KUKA KRL program: EPS_2_25694_LG01A_A_20260223033035.src

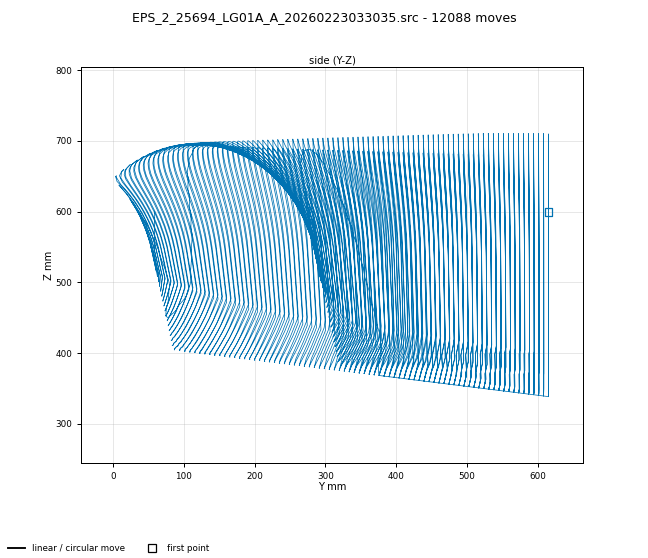
[picture p0: tool path of EPS_2_25694_LG01A_A_20260223033035.src, 12088 of 12090 moves have a stored position in this frame; points joined in program order, loops and branches not executed]
&ACCESS RVP
&REL 4
&COMMENT QRS 19112012
&PARAM EDITMASK = *
DEF PART()
EXT BAS (BAS_COMMAND :IN,REAL :IN )
INT I
BAS (#INITMOV,0 )

;KUKA QRS Post kuka4.cps  Date:22-06-2017 !

File_ID=3040

QRS_PRE_INIT()

;Init var - Until changes are made in qrs_pre_init
Outlet_Square_prg=0
Inlet_1_Square_prg=0
Inlet_2_Square_prg=0
Inlet_3_Square_prg=0
Inlet_4_Square_prg=0
Inlet_5_Square_prg=0

Outlet_1={X 0.000, Y 517.920, Z 561.000, B 0.000, E1 0.000 }
Inlet_1={X 0.000, Y 520.110, Z 531.000, B 0.000, E1 251.000 }
Outlet_1_type=299
Inlet_1_type=299
;QRS#1=Sidecore dimensions
;QRS#2=300-12" PVC SDR 35
;QRS#3=300-12" PVC SDR 35
;QRS#4=
;QRS#5=
;QRS#6=
;QRS#7=
;QRS#8=
;QRS#9=16M PSX
;QRS#10=16M PSX
;QRS#11=
;QRS#12=
;QRS#13=
;QRS#14=
;QRS#15=
;QRS#16=1220x127x991 3,25'
;QRS#17=EPS Height
;QRS#18=710,5
;QRS#19=*
;QRS#20= UPDATED VERSION 22-06-2017
;QRS#21=*
Outlet_Square=0150
Inlet_1_Square=0150
Inlet_2_Square=0
Inlet_3_Square=0
Inlet_4_Square=0
Inlet_5_Square=0
Mill_Square=1
Outlet_Square_Prg=206
Inlet_1_Square_prg=206

QRS_INIT()

$ADVANCE=5

; T1
PTP {E1 173.642,E2 173.642}
PTP {X 0,Y 615.447,A -85,B 0,C 180,E1 173.642,E2 173.642,E3 0,E4 0,E5 0,E6 0}
QRS_SPEED_INIT()
LIN {X 0,Y 615.447,Z 600,A -85,B 0,C 180,E1 173.642,E2 173.642,E3 0,E4 0,E5 0,E6 0} C_VEL
LIN {X 0,Y 615.447,Z 348.502,A -85,B 0,C 180,E1 173.642,E2 173.642} C_VEL
LIN {X 0,Y 615.447,Z 340.324,A -85,B 0,C 180,E1 173.642,E2 173.642} C_VEL
LIN {X 0,Y 615.428,Z 338.324,A -85,B 0,C 180,E1 173.456,E2 173.456} C_VEL
LIN {X 0,Y 615.429,Z 338.324,A -85,B 0,C 180,E1 171.462,E2 171.462} C_VEL
LIN {X 0,Y 615.412,Z 338.324,A -85,B 0,C 180,E1 169.14,E2 169.14} C_VEL
LIN {X 0,Y 615.415,Z 338.325,A -85,B 0,C 180,E1 166.797,E2 166.797} C_VEL
LIN {X 0,Y 615.418,Z 338.324,A -85,B 0,C 180,E1 164.772,E2 164.772} C_VEL
LIN {X 0,Y 615.493,Z 338.326,A -85,B 0,C 180,E1 162.043,E2 162.043} C_VEL
LIN {X 0,Y 615.419,Z 338.323,A -85,B 0,C 180,E1 159.267,E2 159.267} C_VEL
LIN {X 0,Y 615.416,Z 338.323,A -85,B 0,C 180,E1 157.152,E2 157.152} C_VEL
LIN {X 0,Y 615.416,Z 338.323,A -85,B 0,C 180,E1 155.005,E2 155.005} C_VEL
LIN {X 0,Y 615.478,Z 338.329,A -85,B 0,C 180,E1 152.084,E2 152.084} C_VEL
LIN {X 0,Y 615.475,Z 338.321,A -85,B 0,C 180,E1 149.839,E2 149.839} C_VEL
LIN {X 0,Y 615.44,Z 338.322,A -85,B 0,C 180,E1 147.539,E2 147.539} C_VEL
LIN {X 0,Y 615.42,Z 338.322,A -85,B 0,C 180,E1 145.18,E2 145.18} C_VEL
LIN {X 0,Y 615.429,Z 338.323,A -85,B 0,C 180,E1 142.753,E2 142.753} C_VEL
LIN {X 0,Y 615.486,Z 338.32,A -85,B 0,C 180,E1 139.909,E2 139.909} C_VEL
LIN {X 0,Y 615.451,Z 338.32,A -85,B 0,C 180,E1 137.644,E2 137.644} C_VEL
LIN {X 0,Y 615.422,Z 338.322,A -85,B 0,C 180,E1 135.073,E2 135.073} C_VEL
LIN {X 0,Y 615.423,Z 338.322,A -85,B 0,C 180,E1 133.041,E2 133.041} C_VEL
LIN {X 0,Y 615.446,Z 338.323,A -85,B 0,C 180,E1 130.608,E2 130.608} C_VEL
LIN {X 0,Y 615.484,Z 338.322,A -85,B 0,C 180,E1 128.011,E2 128.011} C_VEL
LIN {X 0,Y 615.45,Z 338.319,A -85,B 0,C 180,E1 125.617,E2 125.617} C_VEL
LIN {X 0,Y 615.428,Z 338.32,A -85,B 0,C 180,E1 123.238,E2 123.238} C_VEL
LIN {X 0,Y 615.43,Z 338.322,A -85,B 0,C 180,E1 120.921,E2 120.921} C_VEL
LIN {X 0,Y 615.468,Z 338.325,A -85,B 0,C 180,E1 118.446,E2 118.446} C_VEL
LIN {X 0,Y 615.447,Z 338.318,A -85,B 0,C 180,E1 115.56,E2 115.56} C_VEL
LIN {X 0,Y 615.447,Z 338.318,A -85,B 0,C 180,E1 113.557,E2 113.557} C_VEL
LIN {X 0,Y 615.439,Z 338.319,A -85,B 0,C 180,E1 111.432,E2 111.432} C_VEL
LIN {X 0,Y 615.435,Z 338.319,A -85,B 0,C 180,E1 109.338,E2 109.338} C_VEL
LIN {X 0,Y 615.431,Z 338.32,A -85,B 0,C 180,E1 107.271,E2 107.271} C_VEL
LIN {X 0,Y 615.433,Z 338.319,A -85,B 0,C 180,E1 105.226,E2 105.226} C_VEL
LIN {X 0,Y 615.433,Z 338.32,A -85,B 0,C 180,E1 103.201,E2 103.201} C_VEL
LIN {X 0,Y 615.47,Z 338.324,A -85,B 0,C 180,E1 100.526,E2 100.526} C_VEL
LIN {X 0,Y 615.48,Z 338.315,A -85,B 0,C 180,E1 97.875,E2 97.875} C_VEL
LIN {X 0,Y 615.436,Z 338.319,A -85,B 0,C 180,E1 95.241,E2 95.241} C_VEL
LIN {X 0,Y 615.464,Z 338.323,A -85,B 0,C 180,E1 92.617,E2 92.617} C_VEL
LIN {X 0,Y 615.486,Z 338.316,A -85,B 0,C 180,E1 89.999,E2 89.999} C_VEL
LIN {X 0,Y 615.441,Z 338.317,A -85,B 0,C 180,E1 87.381,E2 87.381} C_VEL
LIN {X 0,Y 615.443,Z 338.317,A -85,B 0,C 180,E1 85.414,E2 85.414} C_VEL
LIN {X 0,Y 615.445,Z 338.317,A -85,B 0,C 180,E1 83.442,E2 83.442} C_VEL
LIN {X 0,Y 615.446,Z 338.316,A -85,B 0,C 180,E1 81.462,E2 81.462} C_VEL
LIN {X 0,Y 615.44,Z 338.319,A -85,B 0,C 180,E1 79.137,E2 79.137} C_VEL
LIN {X 0,Y 615.455,Z 338.322,A -85,B 0,C 180,E1 76.797,E2 76.797} C_VEL
LIN {X 0,Y 615.494,Z 338.315,A -85,B 0,C 180,E1 74.094,E2 74.094} C_VEL
LIN {X 0,Y 615.444,Z 338.317,A -85,B 0,C 180,E1 71.352,E2 71.352} C_VEL
LIN {X 0,Y 615.443,Z 338.318,A -85,B 0,C 180,E1 69.267,E2 69.267} C_VEL
LIN {X 0,Y 615.444,Z 338.319,A -85,B 0,C 180,E1 67.153,E2 67.153} C_VEL
LIN {X 0,Y 615.499,Z 338.325,A -85,B 0,C 180,E1 64.43,E2 64.43} C_VEL
LIN {X 0,Y 615.455,Z 338.315,A -85,B 0,C 180,E1 61.556,E2 61.556} C_VEL
LIN {X 0,Y 615.445,Z 338.32,A -85,B 0,C 180,E1 59.077,E2 59.077} C_VEL
LIN {X 0,Y 615.497,Z 338.325,A -85,B 0,C 180,E1 56.465,E2 56.465} C_VEL
LIN {X 0,Y 615.457,Z 338.314,A -85,B 0,C 180,E1 53.572,E2 53.572} C_VEL
LIN {X 0,Y 615.456,Z 338.32,A -85,B 0,C 180,E1 50.942,E2 50.942} C_VEL
LIN {X 0,Y 615.493,Z 338.326,A -85,B 0,C 180,E1 48.526,E2 48.526} C_VEL
LIN {X 0,Y 615.482,Z 338.311,A -85,B 0,C 180,E1 45.849,E2 45.849} C_VEL
LIN {X 0,Y 615.45,Z 338.317,A -85,B 0,C 180,E1 43.248,E2 43.248} C_VEL
LIN {X 0,Y 615.449,Z 338.397,A -85,B 0,C 180,E1 41.259,E2 41.259} C_VEL
LIN {X 0,Y 615.47,Z 358.127,A -85,B 0,C 180,E1 38.696,E2 38.696} C_VEL
LIN {X 0,Y 615.456,Z 369.9,A -85,B 0,C 180,E1 37.186,E2 37.186} C_VEL
LIN {X 0,Y 615.489,Z 534.997,A -85,B 0,C 180,E1 35.19,E2 35.19} C_VEL
LIN {X 0,Y 615.484,Z 550.512,A -85,B 0,C 180,E1 34.865,E2 34.865} C_VEL
LIN {X 0,Y 615.478,Z 565.792,A -85,B 0,C 180,E1 34.402,E2 34.402} C_VEL
LIN {X 0,Y 615.484,Z 579.854,A -85,B 0,C 180,E1 33.838,E2 33.838} C_VEL
LIN {X 0,Y 615.488,Z 593.728,A -85,B 0,C 180,E1 33.139,E2 33.139} C_VEL
LIN {X 0,Y 615.498,Z 606.785,A -85,B 0,C 180,E1 32.332,E2 32.332} C_VEL
LIN {X 0,Y 615.496,Z 619.457,A -85,B 0,C 180,E1 31.385,E2 31.385} C_VEL
LIN {X 0,Y 615.494,Z 631.006,A -85,B 0,C 180,E1 30.349,E2 30.349} C_VEL
LIN {X 0,Y 615.494,Z 641.505,A -85,B 0,C 180,E1 29.219,E2 29.219} C_VEL
LIN {X 0,Y 615.496,Z 649.597,A -85,B 0,C 180,E1 28.182,E2 28.182} C_VEL
LIN {X 0,Y 615.493,Z 657.085,A -85,B 0,C 180,E1 27.045,E2 27.045} C_VEL
LIN {X 0,Y 615.499,Z 664.276,A -85,B 0,C 180,E1 25.715,E2 25.715} C_VEL
LIN {X 0,Y 615.488,Z 669.041,A -85,B 0,C 180,E1 24.632,E2 24.632} C_VEL
LIN {X 0,Y 615.491,Z 672.806,A -85,B 0,C 180,E1 23.556,E2 23.556} C_VEL
LIN {X 0,Y 615.496,Z 676.516,A -85,B 0,C 180,E1 22.136,E2 22.136} C_VEL
LIN {X 0,Y 615.495,Z 678.815,A -85,B 0,C 180,E1 20.731,E2 20.731} C_VEL
LIN {X 0,Y 615.489,Z 679.804,A -85,B 0,C 180,E1 19.338,E2 19.338} C_VEL
LIN {X 0,Y 615.497,Z 679.524,A -85,B 0,C 180,E1 17.957,E2 17.957} C_VEL
LIN {X 0,Y 615.493,Z 677.757,A -85,B 0,C 180,E1 16.432,E2 16.432} C_VEL
LIN {X 0,Y 615.492,Z 675.277,A -85,B 0,C 180,E1 15.226,E2 15.226} C_VEL
LIN {X 0,Y 615.495,Z 671.262,A -85,B 0,C 180,E1 13.874,E2 13.874} C_VEL
LIN {X 0,Y 615.492,Z 665.885,A -85,B 0,C 180,E1 12.53,E2 12.53} C_VEL
LIN {X 0,Y 615.496,Z 659.043,A -85,B 0,C 180,E1 11.193,E2 11.193} C_VEL
LIN {X 0,Y 615.496,Z 650.583,A -85,B 0,C 180,E1 9.862,E2 9.862} C_VEL
LIN {X 0,Y 615.495,Z 641.592,A -85,B 0,C 180,E1 8.702,E2 8.702} C_VEL
LIN {X 0,Y 615.494,Z 630.85,A -85,B 0,C 180,E1 7.546,E2 7.546} C_VEL
LIN {X 0,Y 615.498,Z 619.859,A -85,B 0,C 180,E1 6.557,E2 6.557} C_VEL
LIN {X 0,Y 615.498,Z 607.894,A -85,B 0,C 180,E1 5.652,E2 5.652} C_VEL
LIN {X 0,Y 615.492,Z 594.819,A -85,B 0,C 180,E1 4.831,E2 4.831} C_VEL
LIN {X 0,Y 615.493,Z 580.329,A -85,B 0,C 180,E1 4.093,E2 4.093} C_VEL
LIN {X 0,Y 615.478,Z 566.113,A -85,B 0,C 180,E1 3.519,E2 3.519} C_VEL
LIN {X 0,Y 615.484,Z 551.397,A -85,B 0,C 180,E1 3.068,E2 3.068} C_VEL
LIN {X 0,Y 615.49,Z 536.141,A -85,B 0,C 180,E1 2.741,E2 2.741} C_VEL
LIN {X 0,Y 615.483,Z 493.536,A -85,B 0,C 180,E1 2.209,E2 2.209} C_VEL
LIN {X 0,Y 615.457,Z 369.836,A -85,B 0,C 180,E1 0.716,E2 0.716} C_VEL
LIN {X 0,Y 615.49,Z 347.76,A -85,B 0,C 180,E1 -2.127,E2 -2.127} C_VEL
LIN {X 0,Y 615.457,Z 338.316,A -85,B 0,C 180,E1 -3.375,E2 -3.375} C_VEL
LIN {X 0,Y 615.487,Z 338.31,A -85,B 0,C 180,E1 -5.898,E2 -5.898} C_VEL
LIN {X 0,Y 615.489,Z 338.327,A -85,B 0,C 180,E1 -8.536,E2 -8.536} C_VEL
LIN {X 0,Y 615.449,Z 338.318,A -85,B 0,C 180,E1 -11.194,E2 -11.194} C_VEL
LIN {X 0,Y 615.491,Z 338.311,A -85,B 0,C 180,E1 -13.933,E2 -13.933} C_VEL
LIN {X 0,Y 615.476,Z 338.325,A -85,B 0,C 180,E1 -16.587,E2 -16.587} C_VEL
LIN {X 0,Y 615.47,Z 338.323,A -85,B 0,C 180,E1 -18.646,E2 -18.646} C_VEL
LIN {X 0,Y 615.458,Z 338.322,A -85,B 0,C 180,E1 -20.732,E2 -20.732} C_VEL
LIN {X 0,Y 615.447,Z 338.322,A -85,B 0,C 180,E1 -22.846,E2 -22.846} C_VEL
LIN {X 0,Y 615.437,Z 338.321,A -85,B 0,C 180,E1 -24.994,E2 -24.994} C_VEL
LIN {X 0,Y 615.432,Z 338.32,A -85,B 0,C 180,E1 -27.18,E2 -27.18} C_VEL
LIN {X 0,Y 615.471,Z 338.317,A -85,B 0,C 180,E1 -29.791,E2 -29.791} C_VEL
LIN {X 0,Y 615.465,Z 338.324,A -85,B 0,C 180,E1 -32.459,E2 -32.459} C_VEL
LIN {X 0,Y 615.43,Z 338.323,A -85,B 0,C 180,E1 -34.819,E2 -34.819} C_VEL
LIN {X 0,Y 615.423,Z 338.322,A -85,B 0,C 180,E1 -37.247,E2 -37.247} C_VEL
LIN {X 0,Y 615.498,Z 338.325,A -85,B 0,C 180,E1 -40.089,E2 -40.089} C_VEL
LIN {X 0,Y 615.457,Z 338.325,A -85,B 0,C 180,E1 -42.355,E2 -42.355} C_VEL
LIN {X 0,Y 615.412,Z 338.325,A -85,B 0,C 180,E1 -44.924,E2 -44.924} C_VEL
LIN {X 0,Y 615.41,Z 338.325,A -85,B 0,C 180,E1 -46.96,E2 -46.96} C_VEL
LIN {X 0,Y 615.426,Z 338.325,A -85,B 0,C 180,E1 -49.388,E2 -49.388} C_VEL
LIN {X 0,Y 615.477,Z 338.328,A -85,B 0,C 180,E1 -51.989,E2 -51.989} C_VEL
LIN {X 0,Y 615.447,Z 338.322,A -85,B 0,C 180,E1 -54.381,E2 -54.381} C_VEL
LIN {X 0,Y 615.423,Z 338.322,A -85,B 0,C 180,E1 -56.759,E2 -56.759} C_VEL
LIN {X 0,Y 615.423,Z 338.323,A -85,B 0,C 180,E1 -59.076,E2 -59.076} C_VEL
LIN {X 0,Y 615.466,Z 338.324,A -85,B 0,C 180,E1 -61.553,E2 -61.553} C_VEL
LIN {X 0,Y 615.447,Z 338.319,A -85,B 0,C 180,E1 -64.439,E2 -64.439} C_VEL
LIN {X 0,Y 615.43,Z 338.439,A -85,B 0,C 180,E1 -64.934,E2 -64.934} C_VEL
LIN {X 0,Y 615.477,Z 359.979,A -85,B 0,C 180,E1 -67.404,E2 -67.404} C_VEL
LIN {X 0,Y 615.49,Z 384.309,A -85,B 0,C 180,E1 -70.141,E2 -70.141} C_VEL
LIN {X 0,Y 615.487,Z 398.969,A -85,B 0,C 180,E1 -71.761,E2 -71.761} C_VEL
LIN {X 0,Y 615.484,Z 565.198,A -85,B 0,C 180,E1 -73.768,E2 -73.768} C_VEL
LIN {X 0,Y 615.49,Z 580.682,A -85,B 0,C 180,E1 -74.094,E2 -74.094} C_VEL
LIN {X 0,Y 615.48,Z 596.028,A -85,B 0,C 180,E1 -74.561,E2 -74.561} C_VEL
LIN {X 0,Y 615.484,Z 609.735,A -85,B 0,C 180,E1 -75.112,E2 -75.112} C_VEL
LIN {X 0,Y 615.493,Z 624.04,A -85,B 0,C 180,E1 -75.833,E2 -75.833} C_VEL
LIN {X 0,Y 615.497,Z 636.886,A -85,B 0,C 180,E1 -76.63,E2 -76.63} C_VEL
LIN {X 0,Y 615.495,Z 649.244,A -85,B 0,C 180,E1 -77.553,E2 -77.553} C_VEL
LIN {X 0,Y 615.495,Z 659.598,A -85,B 0,C 180,E1 -78.473,E2 -78.473} C_VEL
LIN {X 0,Y 615.494,Z 669.176,A -85,B 0,C 180,E1 -79.472,E2 -79.472} C_VEL
LIN {X 0,Y 615.493,Z 678.571,A -85,B 0,C 180,E1 -80.635,E2 -80.635} C_VEL
LIN {X 0,Y 615.497,Z 686.375,A -85,B 0,C 180,E1 -81.793,E2 -81.793} C_VEL
LIN {X 0,Y 615.494,Z 693.607,A -85,B 0,C 180,E1 -83.102,E2 -83.102} C_VEL
LIN {X 0,Y 615.499,Z 699.433,A -85,B 0,C 180,E1 -84.429,E2 -84.429} C_VEL
LIN {X 0,Y 615.491,Z 702.857,A -85,B 0,C 180,E1 -85.415,E2 -85.415} C_VEL
LIN {X 0,Y 615.493,Z 706.316,A -85,B 0,C 180,E1 -86.726,E2 -86.726} C_VEL
LIN {X 0,Y 615.499,Z 708.592,A -85,B 0,C 180,E1 -88.036,E2 -88.036} C_VEL
LIN {X 0,Y 615.491,Z 709.741,A -85,B 0,C 180,E1 -89.345,E2 -89.345} C_VEL
LIN {X 0,Y 615.491,Z 709.741,A -85,B 0,C 180,E1 -90.653,E2 -90.653} C_VEL
LIN {X 0,Y 615.499,Z 708.594,A -85,B 0,C 180,E1 -91.962,E2 -91.962} C_VEL
LIN {X 0,Y 615.493,Z 706.32,A -85,B 0,C 180,E1 -93.272,E2 -93.272} C_VEL
LIN {X 0,Y 615.491,Z 702.863,A -85,B 0,C 180,E1 -94.583,E2 -94.583} C_VEL
LIN {X 0,Y 615.497,Z 698.147,A -85,B 0,C 180,E1 -95.897,E2 -95.897} C_VEL
LIN {X 0,Y 615.492,Z 692.035,A -85,B 0,C 180,E1 -97.215,E2 -97.215} C_VEL
LIN {X 0,Y 615.49,Z 684.34,A -85,B 0,C 180,E1 -98.536,E2 -98.536} C_VEL
LIN {X 0,Y 615.495,Z 676.122,A -85,B 0,C 180,E1 -99.695,E2 -99.695} C_VEL
LIN {X 0,Y 615.496,Z 665.899,A -85,B 0,C 180,E1 -100.892,E2 -100.892} C_VEL
LIN {X 0,Y 615.496,Z 656.079,A -85,B 0,C 180,E1 -101.859,E2 -101.859} C_VEL
LIN {X 0,Y 615.497,Z 643.963,A -85,B 0,C 180,E1 -102.864,E2 -102.864} C_VEL
LIN {X 0,Y 615.498,Z 631.815,A -85,B 0,C 180,E1 -103.704,E2 -103.704} C_VEL
LIN {X 0,Y 615.477,Z 618.398,A -85,B 0,C 180,E1 -104.472,E2 -104.472} C_VEL
LIN {X 0,Y 615.495,Z 603.875,A -85,B 0,C 180,E1 -105.14,E2 -105.14} C_VEL
LIN {X 0,Y 615.48,Z 589.652,A -85,B 0,C 180,E1 -105.649,E2 -105.649} C_VEL
LIN {X 0,Y 615.5,Z 575.193,A -85,B 0,C 180,E1 -106.034,E2 -106.034} C_VEL
LIN {X 0,Y 615.48,Z 560.694,A -85,B 0,C 180,E1 -106.296,E2 -106.296} C_VEL
LIN {X 0,Y 615.489,Z 398.746,A -85,B 0,C 180,E1 -108.258,E2 -108.258} C_VEL
LIN {X 0,Y 615.49,Z 373.403,A -85,B 0,C 180,E1 -111.079,E2 -111.079} C_VEL
LIN {X 0,Y 615.496,Z 347.578,A -85,B 0,C 180,E1 -114.01,E2 -114.01} C_VEL
LIN {X 0,Y 615.43,Z 338.321,A -85,B 0,C 180,E1 -115.099,E2 -115.099} C_VEL
LIN {X 0,Y 615.429,Z 338.32,A -85,B 0,C 180,E1 -117.179,E2 -117.179} C_VEL
LIN {X 0,Y 615.47,Z 338.317,A -85,B 0,C 180,E1 -119.792,E2 -119.792} C_VEL
LIN {X 0,Y 615.468,Z 338.324,A -85,B 0,C 180,E1 -122.457,E2 -122.457} C_VEL
LIN {X 0,Y 615.435,Z 338.322,A -85,B 0,C 180,E1 -124.817,E2 -124.817} C_VEL
LIN {X 0,Y 615.428,Z 338.32,A -85,B 0,C 180,E1 -127.245,E2 -127.245} C_VEL
LIN {X 0,Y 615.499,Z 338.321,A -85,B 0,C 180,E1 -130.09,E2 -130.09} C_VEL
LIN {X 0,Y 615.476,Z 338.324,A -85,B 0,C 180,E1 -132.352,E2 -132.352} C_VEL
LIN {X 0,Y 615.426,Z 338.322,A -85,B 0,C 180,E1 -134.926,E2 -134.926} C_VEL
LIN {X 0,Y 615.425,Z 338.322,A -85,B 0,C 180,E1 -136.957,E2 -136.957} C_VEL
LIN {X 0,Y 615.431,Z 338.321,A -85,B 0,C 180,E1 -139.389,E2 -139.389} C_VEL
LIN {X 0,Y 615.478,Z 338.324,A -85,B 0,C 180,E1 -141.987,E2 -141.987} C_VEL
LIN {X 0,Y 615.465,Z 338.324,A -85,B 0,C 180,E1 -144.383,E2 -144.383} C_VEL
LIN {X 0,Y 615.429,Z 338.323,A -85,B 0,C 180,E1 -146.76,E2 -146.76} C_VEL
LIN {X 0,Y 615.419,Z 338.323,A -85,B 0,C 180,E1 -149.077,E2 -149.077} C_VEL
LIN {X 0,Y 615.425,Z 338.322,A -85,B 0,C 180,E1 -151.339,E2 -151.339} C_VEL
LIN {X 0,Y 615.472,Z 338.325,A -85,B 0,C 180,E1 -154.284,E2 -154.284} C_VEL
LIN {X 0,Y 615.451,Z 338.324,A -85,B 0,C 180,E1 -156.442,E2 -156.442} C_VEL
LIN {X 0,Y 615.437,Z 338.324,A -85,B 0,C 180,E1 -158.566,E2 -158.566} C_VEL
LIN {X 0,Y 615.429,Z 338.324,A -85,B 0,C 180,E1 -160.66,E2 -160.66} C_VEL
LIN {X 0,Y 615.423,Z 338.324,A -85,B 0,C 180,E1 -162.728,E2 -162.728} C_VEL
LIN {X 0,Y 615.42,Z 338.324,A -85,B 0,C 180,E1 -164.772,E2 -164.772} C_VEL
LIN {X 0,Y 615.416,Z 338.325,A -85,B 0,C 180,E1 -166.797,E2 -166.797} C_VEL
LIN {X 0,Y 615.413,Z 338.324,A -85,B 0,C 180,E1 -169.139,E2 -169.139} C_VEL
LIN {X 0,Y 615.429,Z 338.324,A -85,B 0,C 180,E1 -171.463,E2 -171.463} C_VEL
LIN {X 0,Y 615.485,Z 338.326,A -85,B 0,C 180,E1 -174.102,E2 -174.102} C_VEL
LIN {X 0,Y 615.417,Z 338.325,A -85,B 0,C 180,E1 -176.727,E2 -176.727} C_VEL
LIN {X 0,Y 615.418,Z 338.325,A -85,B 0,C 180,E1 -178.691,E2 -178.691} C_VEL
LIN {X 0,Y 615.419,Z 338.325,A -85,B 0,C 180,E1 -180.655,E2 -180.655} C_VEL
LIN {X 0,Y 615.421,Z 338.325,A -85,B 0,C 180,E1 -182.618,E2 -182.618} C_VEL
LIN {X 0,Y 615.424,Z 338.325,A -85,B 0,C 180,E1 -184.585,E2 -184.585} C_VEL
LIN {X 0,Y 615.428,Z 338.324,A -85,B 0,C 180,E1 -186.544,E2 -186.544} C_VEL
LIN {X 0,Y 614.74,Z 338.47,A -85,B 0,C 180,E1 -187.09,E2 -187.09} C_VEL
LIN {X 0,Y 611.894,Z 338.895,A -85,B 0,C 180,E1 -187.976,E2 -187.976} C_VEL
LIN {X 0,Y 609.509,Z 339.197,A -85,B 0,C 180,E1 -188.689,E2 -188.689} C_VEL
LIN {X 0,Y 608.491,Z 339.31,A -85,B 0,C 180,E1 -189.239,E2 -189.239} C_VEL
LIN {X 0,Y 608.411,Z 339.319,A -85,B 0,C 180,E1 -189.425,E2 -189.425} C_VEL
LIN {X 0,Y 608.443,Z 339.324,A -85,B 0,C 180,E1 -192,E2 -192} C_VEL
LIN {X 0,Y 608.389,Z 339.321,A -85,B 0,C 180,E1 -194.723,E2 -194.723} C_VEL
LIN {X 0,Y 608.397,Z 339.319,A -85,B 0,C 180,E1 -196.786,E2 -196.786} C_VEL
LIN {X 0,Y 608.412,Z 339.317,A -85,B 0,C 180,E1 -198.871,E2 -198.871} C_VEL
LIN {X 0,Y 608.436,Z 339.321,A -85,B 0,C 180,E1 -201.693,E2 -201.693} C_VEL
LIN {X 0,Y 608.412,Z 339.318,A -85,B 0,C 180,E1 -204.573,E2 -204.573} C_VEL
LIN {X 0,Y 608.402,Z 339.319,A -85,B 0,C 180,E1 -207.197,E2 -207.197} C_VEL
LIN {X 0,Y 608.462,Z 339.32,A -85,B 0,C 180,E1 -209.974,E2 -209.974} C_VEL
LIN {X 0,Y 608.411,Z 339.317,A -85,B 0,C 180,E1 -212.883,E2 -212.883} C_VEL
LIN {X 0,Y 608.406,Z 339.32,A -85,B 0,C 180,E1 -215.28,E2 -215.28} C_VEL
LIN {X 0,Y 608.451,Z 339.317,A -85,B 0,C 180,E1 -218.241,E2 -218.241} C_VEL
LIN {X 0,Y 608.399,Z 339.32,A -85,B 0,C 180,E1 -221.182,E2 -221.182} C_VEL
LIN {X 0,Y 608.461,Z 339.322,A -85,B 0,C 180,E1 -223.871,E2 -223.871} C_VEL
LIN {X 0,Y 608.421,Z 339.316,A -85,B 0,C 180,E1 -226.697,E2 -226.697} C_VEL
LIN {X 0,Y 608.396,Z 339.319,A -85,B 0,C 180,E1 -228.82,E2 -228.82} C_VEL
LIN {X 0,Y 608.46,Z 339.322,A -85,B 0,C 180,E1 -231.761,E2 -231.761} C_VEL
LIN {X 0,Y 608.405,Z 339.318,A -85,B 0,C 180,E1 -234.722,E2 -234.722} C_VEL
LIN {X 0,Y 608.443,Z 339.319,A -85,B 0,C 180,E1 -237.481,E2 -237.481} C_VEL
LIN {X 0,Y 608.456,Z 339.315,A -85,B 0,C 180,E1 -240.221,E2 -240.221} C_VEL
LIN {X 0,Y 608.411,Z 339.317,A -85,B 0,C 180,E1 -242.806,E2 -242.806} C_VEL
LIN {X 0,Y 608.432,Z 339.32,A -85,B 0,C 180,E1 -245.429,E2 -245.429} C_VEL
LIN {X 0,Y 608.445,Z 339.315,A -85,B 0,C 180,E1 -248.309,E2 -248.309} C_VEL
LIN {X 0,Y 608.432,Z 339.316,A -85,B 0,C 180,E1 -251.131,E2 -251.131} C_VEL
LIN {X 0,Y 608.455,Z 339.319,A -85,B 0,C 180,E1 -253.907,E2 -253.907} C_VEL
LIN {X 0,Y 608.425,Z 339.316,A -85,B 0,C 180,E1 -256.644,E2 -256.644} C_VEL
LIN {X 0,Y 608.439,Z 339.319,A -85,B 0,C 180,E1 -259.351,E2 -259.351} C_VEL
LIN {X 0,Y 608.472,Z 339.315,A -85,B 0,C 180,E1 -262.034,E2 -262.034} C_VEL
LIN {X 0,Y 608.422,Z 339.316,A -85,B 0,C 180,E1 -264.699,E2 -264.699} C_VEL
LIN {X 0,Y 608.456,Z 339.317,A -85,B 0,C 180,E1 -267.353,E2 -267.353} C_VEL
LIN {X 0,Y 608.477,Z 339.314,A -85,B 0,C 180,E1 -270.001,E2 -270.001} C_VEL
LIN {X 0,Y 608.437,Z 339.314,A -85,B 0,C 180,E1 -272.649,E2 -272.649} C_VEL
LIN {X 0,Y 608.44,Z 339.319,A -85,B 0,C 180,E1 -275.303,E2 -275.303} C_VEL
LIN {X 0,Y 608.481,Z 339.313,A -85,B 0,C 180,E1 -277.968,E2 -277.968} C_VEL
LIN {X 0,Y 608.412,Z 339.318,A -85,B 0,C 180,E1 -280.926,E2 -280.926} C_VEL
LIN {X 0,Y 608.444,Z 339.32,A -85,B 0,C 180,E1 -283.358,E2 -283.358} C_VEL
LIN {X 0,Y 608.454,Z 339.315,A -85,B 0,C 180,E1 -286.095,E2 -286.095} C_VEL
LIN {X 0,Y 608.438,Z 339.315,A -85,B 0,C 180,E1 -288.871,E2 -288.871} C_VEL
LIN {X 0,Y 608.466,Z 339.319,A -85,B 0,C 180,E1 -291.692,E2 -291.692} C_VEL
LIN {X 0,Y 608.431,Z 339.315,A -85,B 0,C 180,E1 -294.573,E2 -294.573} C_VEL
LIN {X 0,Y 608.456,Z 339.316,A -85,B 0,C 180,E1 -297.202,E2 -297.202} C_VEL
LIN {X 0,Y 608.471,Z 339.313,A -85,B 0,C 180,E1 -299.971,E2 -299.971} C_VEL
LIN {X 0,Y 608.438,Z 339.315,A -85,B 0,C 180,E1 -302.881,E2 -302.881} C_VEL
LIN {X 0,Y 608.435,Z 339.321,A -85,B 0,C 180,E1 -305.279,E2 -305.279} C_VEL
LIN {X 0,Y 608.461,Z 339.312,A -85,B 0,C 180,E1 -308.239,E2 -308.239} C_VEL
LIN {X 0,Y 608.436,Z 339.32,A -85,B 0,C 180,E1 -311.179,E2 -311.179} C_VEL
LIN {X 0,Y 608.469,Z 339.314,A -85,B 0,C 180,E1 -313.87,E2 -313.87} C_VEL
LIN {X 0,Y 608.443,Z 339.314,A -85,B 0,C 180,E1 -316.695,E2 -316.695} C_VEL
LIN {X 0,Y 608.452,Z 339.413,A -85,B 0,C 180,E1 -318.605,E2 -318.605} C_VEL
LIN {X 0,Y 608.56,Z 355.829,A -85,B 0,C 180,E1 -320.769,E2 -320.769} C_VEL
LIN {X 0,Y 608.514,Z 369.959,A -85,B 0,C 180,E1 -322.602,E2 -322.602} C_VEL
LIN {X 0,Y 608.722,Z 389.584,A -85,B 0,C 180,E1 -322.847,E2 -322.847} C_VEL
LIN {X 0,Y 608.681,Z 535.005,A -85,B 0,C 180,E1 -324.624,E2 -324.624} C_VEL
LIN {X 0,Y 608.662,Z 550.554,A -85,B 0,C 180,E1 -324.953,E2 -324.953} C_VEL
LIN {X 0,Y 608.622,Z 565.582,A -85,B 0,C 180,E1 -325.412,E2 -325.412} C_VEL
LIN {X 0,Y 608.593,Z 579.847,A -85,B 0,C 180,E1 -325.989,E2 -325.989} C_VEL
LIN {X 0,Y 608.56,Z 594.378,A -85,B 0,C 180,E1 -326.732,E2 -326.732} C_VEL
LIN {X 0,Y 608.548,Z 607.869,A -85,B 0,C 180,E1 -327.582,E2 -327.582} C_VEL
LIN {X 0,Y 608.502,Z 620.973,A -85,B 0,C 180,E1 -328.588,E2 -328.588} C_VEL
LIN {X 0,Y 608.49,Z 632.126,A -85,B 0,C 180,E1 -329.616,E2 -329.616} C_VEL
LIN {X 0,Y 608.473,Z 642.777,A -85,B 0,C 180,E1 -330.791,E2 -330.791} C_VEL
LIN {X 0,Y 608.45,Z 651.385,A -85,B 0,C 180,E1 -331.921,E2 -331.921} C_VEL
LIN {X 0,Y 608.439,Z 659.596,A -85,B 0,C 180,E1 -333.225,E2 -333.225} C_VEL
LIN {X 0,Y 608.436,Z 665.098,A -85,B 0,C 180,E1 -334.287,E2 -334.287} C_VEL
LIN {X 0,Y 608.421,Z 669.988,A -85,B 0,C 180,E1 -335.427,E2 -335.427} C_VEL
LIN {X 0,Y 608.435,Z 674.764,A -85,B 0,C 180,E1 -336.875,E2 -336.875} C_VEL
LIN {X 0,Y 608.421,Z 678.035,A -85,B 0,C 180,E1 -338.306,E2 -338.306} C_VEL
LIN {X 0,Y 608.434,Z 679.915,A -85,B 0,C 180,E1 -339.725,E2 -339.725} C_VEL
LIN {X 0,Y 608.425,Z 680.486,A -85,B 0,C 180,E1 -341.129,E2 -341.129} C_VEL
LIN {X 0,Y 608.417,Z 679.79,A -85,B 0,C 180,E1 -342.522,E2 -342.522} C_VEL
LIN {X 0,Y 608.432,Z 677.832,A -85,B 0,C 180,E1 -343.905,E2 -343.905} C_VEL
LIN {X 0,Y 608.416,Z 674.596,A -85,B 0,C 180,E1 -345.278,E2 -345.278} C_VEL
LIN {X 0,Y 608.441,Z 670.061,A -85,B 0,C 180,E1 -346.643,E2 -346.643} C_VEL
LIN {X 0,Y 608.437,Z 664.145,A -85,B 0,C 180,E1 -348,E2 -348} C_VEL
LIN {X 0,Y 608.44,Z 656.711,A -85,B 0,C 180,E1 -349.35,E2 -349.35} C_VEL
LIN {X 0,Y 608.479,Z 648.796,A -85,B 0,C 180,E1 -350.526,E2 -350.526} C_VEL
LIN {X 0,Y 608.494,Z 639.349,A -85,B 0,C 180,E1 -351.699,E2 -351.699} C_VEL
LIN {X 0,Y 608.493,Z 628.05,A -85,B 0,C 180,E1 -352.868,E2 -352.868} C_VEL
LIN {X 0,Y 608.539,Z 616.453,A -85,B 0,C 180,E1 -353.867,E2 -353.867} C_VEL
LIN {X 0,Y 608.551,Z 603.758,A -85,B 0,C 180,E1 -354.782,E2 -354.782} C_VEL
LIN {X 0,Y 608.58,Z 591.256,A -85,B 0,C 180,E1 -355.529,E2 -355.529} C_VEL
LIN {X 0,Y 608.596,Z 577.743,A -85,B 0,C 180,E1 -356.193,E2 -356.193} C_VEL
LIN {X 0,Y 608.622,Z 562.746,A -85,B 0,C 180,E1 -356.773,E2 -356.773} C_VEL
LIN {X 0,Y 608.669,Z 547.601,A -85,B 0,C 180,E1 -357.208,E2 -357.208} C_VEL
LIN {X 0,Y 608.686,Z 532.863,A -85,B 0,C 180,E1 -357.498,E2 -357.498} C_VEL
LIN {X 0,Y 608.67,Z 370.852,A -85,B 0,C 180,E1 -359.473,E2 -359.473} C_VEL
LIN {X 0,Y 608.507,Z 369.83,A -85,B 0,C 180,E1 -359.504,E2 -359.504} C_VEL
LIN {X 0,Y 608.581,Z 348.227,A -85,B 0,C 180,E1 -362.316,E2 -362.316} C_VEL
LIN {X 0,Y 608.44,Z 339.316,A -85,B 0,C 180,E1 -363.518,E2 -363.518} C_VEL
LIN {X 0,Y 608.461,Z 339.313,A -85,B 0,C 180,E1 -365.967,E2 -365.967} C_VEL
LIN {X 0,Y 608.454,Z 339.322,A -85,B 0,C 180,E1 -368.636,E2 -368.636} C_VEL
LIN {X 0,Y 608.427,Z 339.316,A -85,B 0,C 180,E1 -371.325,E2 -371.325} C_VEL
LIN {X 0,Y 608.474,Z 339.313,A -85,B 0,C 180,E1 -374.037,E2 -374.037} C_VEL
LIN {X 0,Y 608.432,Z 339.32,A -85,B 0,C 180,E1 -376.784,E2 -376.784} C_VEL
LIN {X 0,Y 608.428,Z 339.316,A -85,B 0,C 180,E1 -379.571,E2 -379.571} C_VEL
LIN {X 0,Y 608.463,Z 339.32,A -85,B 0,C 180,E1 -382.476,E2 -382.476} C_VEL
LIN {X 0,Y 608.438,Z 339.32,A -85,B 0,C 180,E1 -384.572,E2 -384.572} C_VEL
LIN {X 0,Y 608.416,Z 339.317,A -85,B 0,C 180,E1 -387.195,E2 -387.195} C_VEL
LIN {X 0,Y 608.462,Z 339.317,A -85,B 0,C 180,E1 -389.97,E2 -389.97} C_VEL
LIN {X 0,Y 608.422,Z 339.317,A -85,B 0,C 180,E1 -392.882,E2 -392.882} C_VEL
LIN {X 0,Y 608.405,Z 339.318,A -85,B 0,C 180,E1 -395.28,E2 -395.28} C_VEL
LIN {X 0,Y 608.461,Z 339.32,A -85,B 0,C 180,E1 -398.239,E2 -398.239} C_VEL
LIN {X 0,Y 608.436,Z 339.321,A -85,B 0,C 180,E1 -400.326,E2 -400.326} C_VEL
LIN {X 0,Y 608.43,Z 339.321,A -85,B 0,C 180,E1 -402.33,E2 -402.33} C_VEL
LIN {X 0,Y 608.396,Z 339.32,A -85,B 0,C 180,E1 -404.801,E2 -404.801} C_VEL
LIN {X 0,Y 608.382,Z 339.321,A -85,B 0,C 180,E1 -407.033,E2 -407.033} C_VEL
LIN {X 0,Y 608.384,Z 339.321,A -85,B 0,C 180,E1 -408.817,E2 -408.817} C_VEL
LIN {X 0,Y 608.401,Z 339.319,A -85,B 0,C 180,E1 -410.71,E2 -410.71} C_VEL
LIN {X 0,Y 608.389,Z 339.321,A -85,B 0,C 180,E1 -413.08,E2 -413.08} C_VEL
LIN {X 0,Y 608.437,Z 339.319,A -85,B 0,C 180,E1 -415.528,E2 -415.528} C_VEL
LIN {X 0,Y 608.45,Z 339.323,A -85,B 0,C 180,E1 -417.904,E2 -417.904} C_VEL
LIN {X 0,Y 608.456,Z 339.316,A -85,B 0,C 180,E1 -420.219,E2 -420.219} C_VEL
LIN {X 0,Y 608.412,Z 339.318,A -85,B 0,C 180,E1 -422.805,E2 -422.805} C_VEL
LIN {X 0,Y 608.436,Z 339.441,A -85,B 0,C 180,E1 -424.743,E2 -424.743} C_VEL
LIN {X 0,Y 608.662,Z 351.536,A -85,B 0,C 180,E1 -426.162,E2 -426.162} C_VEL
LIN {X 0,Y 608.595,Z 374.945,A -85,B 0,C 180,E1 -428.845,E2 -428.845} C_VEL
LIN {X 0,Y 608.576,Z 398.969,A -85,B 0,C 180,E1 -431.546,E2 -431.546} C_VEL
LIN {X 0,Y 608.708,Z 508.213,A -85,B 0,C 180,E1 -432.877,E2 -432.877} C_VEL
LIN {X 0,Y 608.679,Z 565.198,A -85,B 0,C 180,E1 -433.582,E2 -433.582} C_VEL
LIN {X 0,Y 608.651,Z 580.681,A -85,B 0,C 180,E1 -433.911,E2 -433.911} C_VEL
LIN {X 0,Y 608.618,Z 596.027,A -85,B 0,C 180,E1 -434.382,E2 -434.382} C_VEL
LIN {X 0,Y 608.605,Z 609.737,A -85,B 0,C 180,E1 -434.94,E2 -434.94} C_VEL
LIN {X 0,Y 608.573,Z 623.221,A -85,B 0,C 180,E1 -435.623,E2 -435.623} C_VEL
LIN {X 0,Y 608.554,Z 635.652,A -85,B 0,C 180,E1 -436.39,E2 -436.39} C_VEL
LIN {X 0,Y 608.528,Z 648.272,A -85,B 0,C 180,E1 -437.323,E2 -437.323} C_VEL
LIN {X 0,Y 608.496,Z 659.739,A -85,B 0,C 180,E1 -438.338,E2 -438.338} C_VEL
LIN {X 0,Y 608.475,Z 669.38,A -85,B 0,C 180,E1 -439.349,E2 -439.349} C_VEL
LIN {X 0,Y 608.477,Z 678.847,A -85,B 0,C 180,E1 -440.526,E2 -440.526} C_VEL
LIN {X 0,Y 608.457,Z 686.724,A -85,B 0,C 180,E1 -441.698,E2 -441.698} C_VEL
LIN {X 0,Y 608.44,Z 694.083,A -85,B 0,C 180,E1 -443.033,E2 -443.033} C_VEL
LIN {X 0,Y 608.45,Z 699.92,A -85,B 0,C 180,E1 -444.365,E2 -444.365} C_VEL
LIN {X 0,Y 608.427,Z 703.38,A -85,B 0,C 180,E1 -445.361,E2 -445.361} C_VEL
LIN {X 0,Y 608.421,Z 706.884,A -85,B 0,C 180,E1 -446.688,E2 -446.688} C_VEL
LIN {X 0,Y 608.444,Z 709.19,A -85,B 0,C 180,E1 -448.013,E2 -448.013} C_VEL
LIN {X 0,Y 608.434,Z 710.35,A -85,B 0,C 180,E1 -449.337,E2 -449.337} C_VEL
LIN {X 0,Y 608.434,Z 710.351,A -85,B 0,C 180,E1 -450.661,E2 -450.661} C_VEL
LIN {X 0,Y 608.444,Z 709.192,A -85,B 0,C 180,E1 -451.985,E2 -451.985} C_VEL
LIN {X 0,Y 608.421,Z 706.888,A -85,B 0,C 180,E1 -453.31,E2 -453.31} C_VEL
LIN {X 0,Y 608.427,Z 703.386,A -85,B 0,C 180,E1 -454.637,E2 -454.637} C_VEL
LIN {X 0,Y 608.435,Z 698.612,A -85,B 0,C 180,E1 -455.966,E2 -455.966} C_VEL
LIN {X 0,Y 608.456,Z 692.432,A -85,B 0,C 180,E1 -457.298,E2 -457.298} C_VEL
LIN {X 0,Y 608.464,Z 684.661,A -85,B 0,C 180,E1 -458.635,E2 -458.635} C_VEL
LIN {X 0,Y 608.471,Z 676.379,A -85,B 0,C 180,E1 -459.808,E2 -459.808} C_VEL
LIN {X 0,Y 608.491,Z 665.657,A -85,B 0,C 180,E1 -461.062,E2 -461.062} C_VEL
LIN {X 0,Y 608.523,Z 654.287,A -85,B 0,C 180,E1 -462.167,E2 -462.167} C_VEL
LIN {X 0,Y 608.547,Z 642.87,A -85,B 0,C 180,E1 -463.098,E2 -463.098} C_VEL
LIN {X 0,Y 608.56,Z 630.466,A -85,B 0,C 180,E1 -463.949,E2 -463.949} C_VEL
LIN {X 0,Y 608.586,Z 616.883,A -85,B 0,C 180,E1 -464.717,E2 -464.717} C_VEL
LIN {X 0,Y 608.631,Z 602.822,A -85,B 0,C 180,E1 -465.358,E2 -465.358} C_VEL
LIN {X 0,Y 608.634,Z 588.34,A -85,B 0,C 180,E1 -465.873,E2 -465.873} C_VEL
LIN {X 0,Y 608.682,Z 573.078,A -85,B 0,C 180,E1 -466.268,E2 -466.268} C_VEL
LIN {X 0,Y 608.681,Z 557.197,A -85,B 0,C 180,E1 -466.533,E2 -466.533} C_VEL
LIN {X 0,Y 608.685,Z 399.699,A -85,B 0,C 180,E1 -468.441,E2 -468.441} C_VEL
LIN {X 0,Y 608.543,Z 398.571,A -85,B 0,C 180,E1 -468.494,E2 -468.494} C_VEL
LIN {X 0,Y 608.617,Z 373.403,A -85,B 0,C 180,E1 -471.329,E2 -471.329} C_VEL
LIN {X 0,Y 608.682,Z 348.444,A -85,B 0,C 180,E1 -474.195,E2 -474.195} C_VEL
LIN {X 0,Y 608.428,Z 339.318,A -85,B 0,C 180,E1 -475.278,E2 -475.278} C_VEL
LIN {X 0,Y 608.437,Z 339.325,A -85,B 0,C 180,E1 -478.266,E2 -478.266} C_VEL
LIN {X 0,Y 608.45,Z 339.318,A -85,B 0,C 180,E1 -480.544,E2 -480.544} C_VEL
LIN {X 0,Y 608.423,Z 339.317,A -85,B 0,C 180,E1 -482.88,E2 -482.88} C_VEL
LIN {X 0,Y 608.406,Z 339.318,A -85,B 0,C 180,E1 -485.278,E2 -485.278} C_VEL
LIN {X 0,Y 608.459,Z 339.322,A -85,B 0,C 180,E1 -488.239,E2 -488.239} C_VEL
LIN {X 0,Y 608.397,Z 339.319,A -85,B 0,C 180,E1 -491.179,E2 -491.179} C_VEL
LIN {X 0,Y 608.421,Z 339.316,A -85,B 0,C 180,E1 -493.304,E2 -493.304} C_VEL
LIN {X 0,Y 608.461,Z 339.321,A -85,B 0,C 180,E1 -496.13,E2 -496.13} C_VEL
LIN {X 0,Y 608.4,Z 339.32,A -85,B 0,C 180,E1 -498.819,E2 -498.819} C_VEL
LIN {X 0,Y 608.449,Z 339.317,A -85,B 0,C 180,E1 -501.759,E2 -501.759} C_VEL
LIN {X 0,Y 608.408,Z 339.32,A -85,B 0,C 180,E1 -504.72,E2 -504.72} C_VEL
LIN {X 0,Y 608.411,Z 339.317,A -85,B 0,C 180,E1 -507.118,E2 -507.118} C_VEL
LIN {X 0,Y 608.463,Z 339.32,A -85,B 0,C 180,E1 -510.026,E2 -510.026} C_VEL
LIN {X 0,Y 608.403,Z 339.319,A -85,B 0,C 180,E1 -512.803,E2 -512.803} C_VEL
LIN {X 0,Y 608.413,Z 339.318,A -85,B 0,C 180,E1 -515.427,E2 -515.427} C_VEL
LIN {X 0,Y 608.437,Z 339.321,A -85,B 0,C 180,E1 -518.307,E2 -518.307} C_VEL
LIN {X 0,Y 608.412,Z 339.317,A -85,B 0,C 180,E1 -521.129,E2 -521.129} C_VEL
LIN {X 0,Y 608.441,Z 339.321,A -85,B 0,C 180,E1 -523.906,E2 -523.906} C_VEL
LIN {X 0,Y 608.413,Z 339.319,A -85,B 0,C 180,E1 -526.643,E2 -526.643} C_VEL
LIN {X 0,Y 608.383,Z 339.321,A -85,B 0,C 180,E1 -529.077,E2 -529.077} C_VEL
LIN {X 0,Y 608.402,Z 339.32,A -85,B 0,C 180,E1 -531.363,E2 -531.363} C_VEL
LIN {X 0,Y 608.475,Z 339.321,A -85,B 0,C 180,E1 -534.033,E2 -534.033} C_VEL
LIN {X 0,Y 608.389,Z 339.321,A -85,B 0,C 180,E1 -536.689,E2 -536.689} C_VEL
LIN {X 0,Y 608.408,Z 339.319,A -85,B 0,C 180,E1 -538.676,E2 -538.676} C_VEL
LIN {X 0,Y 608.397,Z 339.32,A -85,B 0,C 180,E1 -540.662,E2 -540.662} C_VEL
LIN {X 0,Y 608.416,Z 339.318,A -85,B 0,C 180,E1 -542.648,E2 -542.648} C_VEL
LIN {X 0,Y 608.403,Z 339.319,A -85,B 0,C 180,E1 -545.303,E2 -545.303} C_VEL
LIN {X 0,Y 608.461,Z 339.322,A -85,B 0,C 180,E1 -547.967,E2 -547.967} C_VEL
LIN {X 0,Y 608.411,Z 339.319,A -85,B 0,C 180,E1 -549.425,E2 -549.425} C_VEL
LIN {X 0,Y 607.758,Z 339.41,A -85,B 0,C 180,E1 -549.978,E2 -549.978} C_VEL
LIN {X 0,Y 604.927,Z 339.764,A -85,B 0,C 180,E1 -550.875,E2 -550.875} C_VEL
LIN {X 0,Y 602.517,Z 340.063,A -85,B 0,C 180,E1 -551.596,E2 -551.596} C_VEL
LIN {X 0,Y 601.462,Z 340.191,A -85,B 0,C 180,E1 -552.152,E2 -552.152} C_VEL
LIN {X 0,Y 601.366,Z 340.199,A -85,B 0,C 180,E1 -552.341,E2 -552.341} C_VEL
LIN {X 0,Y 601.362,Z 340.195,A -85,B 0,C 180,E1 -554.899,E2 -554.899} C_VEL
LIN {X 0,Y 601.356,Z 340.196,A -85,B 0,C 180,E1 -556.988,E2 -556.988} C_VEL
LIN {X 0,Y 601.384,Z 340.193,A -85,B 0,C 180,E1 -559.1,E2 -559.1} C_VEL
LIN {X 0,Y 601.374,Z 340.204,A -85,B 0,C 180,E1 -561.961,E2 -561.961} C_VEL
LIN {X 0,Y 601.404,Z 340.195,A -85,B 0,C 180,E1 -564.29,E2 -564.29} C_VEL
LIN {X 0,Y 601.363,Z 340.196,A -85,B 0,C 180,E1 -567.116,E2 -567.116} C_VEL
LIN {X 0,Y 601.393,Z 340.197,A -85,B 0,C 180,E1 -570.166,E2 -570.166} C_VEL
LIN {X 0,Y 601.382,Z 340.193,A -85,B 0,C 180,E1 -572.712,E2 -572.712} C_VEL
LIN {X 0,Y 601.351,Z 340.197,A -85,B 0,C 180,E1 -575.109,E2 -575.109} C_VEL
LIN {X 0,Y 601.385,Z 340.196,A -85,B 0,C 180,E1 -577.423,E2 -577.423} C_VEL
LIN {X 0,Y 601.387,Z 340.2,A -85,B 0,C 180,E1 -579.997,E2 -579.997} C_VEL
LIN {X 0,Y 601.354,Z 340.197,A -85,B 0,C 180,E1 -582.676,E2 -582.676} C_VEL
LIN {X 0,Y 601.39,Z 340.197,A -85,B 0,C 180,E1 -585.481,E2 -585.481} C_VEL
LIN {X 0,Y 601.398,Z 340.193,A -85,B 0,C 180,E1 -588.41,E2 -588.41} C_VEL
LIN {X 0,Y 601.371,Z 340.194,A -85,B 0,C 180,E1 -590.872,E2 -590.872} C_VEL
LIN {X 0,Y 601.384,Z 340.203,A -85,B 0,C 180,E1 -593.742,E2 -593.742} C_VEL
LIN {X 0,Y 601.399,Z 340.191,A -85,B 0,C 180,E1 -596.686,E2 -596.686} C_VEL
LIN {X 0,Y 601.393,Z 340.192,A -85,B 0,C 180,E1 -599.058,E2 -599.058} C_VEL
LIN {X 0,Y 601.38,Z 340.197,A -85,B 0,C 180,E1 -601.372,E2 -601.372} C_VEL
LIN {X 0,Y 601.389,Z 340.194,A -85,B 0,C 180,E1 -604.382,E2 -604.382} C_VEL
LIN {X 0,Y 601.373,Z 340.194,A -85,B 0,C 180,E1 -606.589,E2 -606.589} C_VEL
LIN {X 0,Y 601.414,Z 340.195,A -85,B 0,C 180,E1 -609.479,E2 -609.479} C_VEL
LIN {X 0,Y 601.374,Z 340.196,A -85,B 0,C 180,E1 -612.312,E2 -612.312} C_VEL
LIN {X 0,Y 601.387,Z 340.193,A -85,B 0,C 180,E1 -614.409,E2 -614.409} C_VEL
LIN {X 0,Y 601.391,Z 340.192,A -85,B 0,C 180,E1 -616.485,E2 -616.485} C_VEL
LIN {X 0,Y 601.379,Z 340.196,A -85,B 0,C 180,E1 -619.224,E2 -619.224} C_VEL
LIN {X 0,Y 601.434,Z 340.193,A -85,B 0,C 180,E1 -621.94,E2 -621.94} C_VEL
LIN {X 0,Y 601.392,Z 340.192,A -85,B 0,C 180,E1 -624.637,E2 -624.637} C_VEL
LIN {X 0,Y 601.421,Z 340.193,A -85,B 0,C 180,E1 -627.322,E2 -627.322} C_VEL
LIN {X 0,Y 601.445,Z 340.19,A -85,B 0,C 180,E1 -630.001,E2 -630.001} C_VEL
LIN {X 0,Y 601.406,Z 340.19,A -85,B 0,C 180,E1 -632.68,E2 -632.68} C_VEL
LIN {X 0,Y 601.408,Z 340.196,A -85,B 0,C 180,E1 -635.365,E2 -635.365} C_VEL
LIN {X 0,Y 601.439,Z 340.189,A -85,B 0,C 180,E1 -638.062,E2 -638.062} C_VEL
LIN {X 0,Y 601.39,Z 340.194,A -85,B 0,C 180,E1 -640.993,E2 -640.993} C_VEL
LIN {X 0,Y 601.406,Z 340.199,A -85,B 0,C 180,E1 -643.517,E2 -643.517} C_VEL
LIN {X 0,Y 601.412,Z 340.19,A -85,B 0,C 180,E1 -646.288,E2 -646.288} C_VEL
LIN {X 0,Y 601.409,Z 340.192,A -85,B 0,C 180,E1 -649.1,E2 -649.1} C_VEL
LIN {X 0,Y 601.4,Z 340.195,A -85,B 0,C 180,E1 -651.96,E2 -651.96} C_VEL
LIN {X 0,Y 601.388,Z 340.193,A -85,B 0,C 180,E1 -654.88,E2 -654.88} C_VEL
LIN {X 0,Y 601.401,Z 340.198,A -85,B 0,C 180,E1 -657.359,E2 -657.359} C_VEL
LIN {X 0,Y 601.41,Z 340.191,A -85,B 0,C 180,E1 -660.166,E2 -660.166} C_VEL
LIN {X 0,Y 601.402,Z 340.191,A -85,B 0,C 180,E1 -662.712,E2 -662.712} C_VEL
LIN {X 0,Y 601.378,Z 340.197,A -85,B 0,C 180,E1 -665.109,E2 -665.109} C_VEL
LIN {X 0,Y 601.435,Z 340.196,A -85,B 0,C 180,E1 -667.42,E2 -667.42} C_VEL
LIN {X 0,Y 601.405,Z 340.193,A -85,B 0,C 180,E1 -669.996,E2 -669.996} C_VEL
LIN {X 0,Y 601.376,Z 340.194,A -85,B 0,C 180,E1 -672.674,E2 -672.674} C_VEL
LIN {X 0,Y 601.403,Z 340.191,A -85,B 0,C 180,E1 -674.533,E2 -674.533} C_VEL
LIN {X 0,Y 601.413,Z 340.2,A -85,B 0,C 180,E1 -677.41,E2 -677.41} C_VEL
LIN {X 0,Y 601.447,Z 340.386,A -85,B 0,C 180,E1 -678.46,E2 -678.46} C_VEL
LIN {X 0,Y 601.655,Z 350.452,A -85,B 0,C 180,E1 -679.813,E2 -679.813} C_VEL
LIN {X 0,Y 601.562,Z 369.975,A -85,B 0,C 180,E1 -682.381,E2 -682.381} C_VEL
LIN {X 0,Y 601.991,Z 373.736,A -85,B 0,C 180,E1 -682.441,E2 -682.441} C_VEL
LIN {X 0,Y 601.875,Z 535.229,A -85,B 0,C 180,E1 -684.437,E2 -684.437} C_VEL
LIN {X 0,Y 601.843,Z 550.636,A -85,B 0,C 180,E1 -684.767,E2 -684.767} C_VEL
LIN {X 0,Y 601.767,Z 565.987,A -85,B 0,C 180,E1 -685.244,E2 -685.244} C_VEL
LIN {X 0,Y 601.694,Z 580.601,A -85,B 0,C 180,E1 -685.848,E2 -685.848} C_VEL
LIN {X 0,Y 601.643,Z 595.015,A -85,B 0,C 180,E1 -686.6,E2 -686.6} C_VEL
LIN {X 0,Y 601.575,Z 608.835,A -85,B 0,C 180,E1 -687.493,E2 -687.493} C_VEL
LIN {X 0,Y 601.521,Z 620.982,A -85,B 0,C 180,E1 -688.442,E2 -688.442} C_VEL
LIN {X 0,Y 601.488,Z 631.834,A -85,B 0,C 180,E1 -689.451,E2 -689.451} C_VEL
LIN {X 0,Y 601.445,Z 642.289,A -85,B 0,C 180,E1 -690.608,E2 -690.608} C_VEL
LIN {X 0,Y 601.382,Z 650.966,A -85,B 0,C 180,E1 -691.751,E2 -691.751} C_VEL
LIN {X 0,Y 601.37,Z 659.271,A -85,B 0,C 180,E1 -693.073,E2 -693.073} C_VEL
LIN {X 0,Y 601.344,Z 665.916,A -85,B 0,C 180,E1 -694.378,E2 -694.378} C_VEL
LIN {X 0,Y 601.325,Z 671.357,A -85,B 0,C 180,E1 -695.732,E2 -695.732} C_VEL
LIN {X 0,Y 601.325,Z 674.117,A -85,B 0,C 180,E1 -696.586,E2 -696.586} C_VEL
LIN {X 0,Y 601.341,Z 677.615,A -85,B 0,C 180,E1 -698.038,E2 -698.038} C_VEL
LIN {X 0,Y 601.35,Z 679.706,A -85,B 0,C 180,E1 -699.475,E2 -699.475} C_VEL
LIN {X 0,Y 601.312,Z 680.472,A -85,B 0,C 180,E1 -700.897,E2 -700.897} C_VEL
LIN {X 0,Y 601.31,Z 679.968,A -85,B 0,C 180,E1 -702.309,E2 -702.309} C_VEL
LIN {X 0,Y 601.346,Z 678.211,A -85,B 0,C 180,E1 -703.71,E2 -703.71} C_VEL
LIN {X 0,Y 601.313,Z 675.197,A -85,B 0,C 180,E1 -705.1,E2 -705.1} C_VEL
LIN {X 0,Y 601.339,Z 670.899,A -85,B 0,C 180,E1 -706.482,E2 -706.482} C_VEL
LIN {X 0,Y 601.372,Z 665.227,A -85,B 0,C 180,E1 -707.856,E2 -707.856} C_VEL
LIN {X 0,Y 601.364,Z 658.057,A -85,B 0,C 180,E1 -709.223,E2 -709.223} C_VEL
LIN {X 0,Y 601.4,Z 650.442,A -85,B 0,C 180,E1 -710.414,E2 -710.414} C_VEL
LIN {X 0,Y 601.456,Z 641.298,A -85,B 0,C 180,E1 -711.601,E2 -711.601} C_VEL
LIN {X 0,Y 601.472,Z 630.376,A -85,B 0,C 180,E1 -712.784,E2 -712.784} C_VEL
LIN {X 0,Y 601.53,Z 618.407,A -85,B 0,C 180,E1 -713.861,E2 -713.861} C_VEL
LIN {X 0,Y 601.579,Z 605.821,A -85,B 0,C 180,E1 -714.805,E2 -714.805} C_VEL
LIN {X 0,Y 601.653,Z 592.246,A -85,B 0,C 180,E1 -715.645,E2 -715.645} C_VEL
LIN {X 0,Y 601.73,Z 578.95,A -85,B 0,C 180,E1 -716.317,E2 -716.317} C_VEL
LIN {X 0,Y 601.774,Z 564.33,A -85,B 0,C 180,E1 -716.904,E2 -716.904} C_VEL
LIN {X 0,Y 601.86,Z 548.922,A -85,B 0,C 180,E1 -717.364,E2 -717.364} C_VEL
LIN {X 0,Y 601.893,Z 533.575,A -85,B 0,C 180,E1 -717.679,E2 -717.679} C_VEL
LIN {X 0,Y 601.912,Z 371.771,A -85,B 0,C 180,E1 -719.676,E2 -719.676} C_VEL
LIN {X 0,Y 601.552,Z 369.806,A -85,B 0,C 180,E1 -719.728,E2 -719.728} C_VEL
LIN {X 0,Y 601.677,Z 348.693,A -85,B 0,C 180,E1 -722.51,E2 -722.51} C_VEL
LIN {X 0,Y 601.42,Z 340.299,A -85,B 0,C 180,E1 -723.643,E2 -723.643} C_VEL
LIN {X 0,Y 601.413,Z 340.193,A -85,B 0,C 180,E1 -726.037,E2 -726.037} C_VEL
LIN {X 0,Y 601.411,Z 340.197,A -85,B 0,C 180,E1 -728.738,E2 -728.738} C_VEL
LIN {X 0,Y 601.407,Z 340.19,A -85,B 0,C 180,E1 -731.458,E2 -731.458} C_VEL
LIN {X 0,Y 601.423,Z 340.194,A -85,B 0,C 180,E1 -734.205,E2 -734.205} C_VEL
LIN {X 0,Y 601.404,Z 340.193,A -85,B 0,C 180,E1 -736.987,E2 -736.987} C_VEL
LIN {X 0,Y 601.392,Z 340.194,A -85,B 0,C 180,E1 -739.81,E2 -739.81} C_VEL
LIN {X 0,Y 601.41,Z 340.195,A -85,B 0,C 180,E1 -742.683,E2 -742.683} C_VEL
LIN {X 0,Y 601.379,Z 340.196,A -85,B 0,C 180,E1 -744.879,E2 -744.879} C_VEL
LIN {X 0,Y 601.373,Z 340.194,A -85,B 0,C 180,E1 -747.354,E2 -747.354} C_VEL
LIN {X 0,Y 601.407,Z 340.2,A -85,B 0,C 180,E1 -750.165,E2 -750.165} C_VEL
LIN {X 0,Y 601.4,Z 340.194,A -85,B 0,C 180,E1 -752.711,E2 -752.711} C_VEL
LIN {X 0,Y 601.355,Z 340.197,A -85,B 0,C 180,E1 -755.106,E2 -755.106} C_VEL
LIN {X 0,Y 601.384,Z 340.194,A -85,B 0,C 180,E1 -757.423,E2 -757.423} C_VEL
LIN {X 0,Y 601.395,Z 340.201,A -85,B 0,C 180,E1 -759.996,E2 -759.996} C_VEL
LIN {X 0,Y 601.352,Z 340.199,A -85,B 0,C 180,E1 -762.675,E2 -762.675} C_VEL
LIN {X 0,Y 601.369,Z 340.198,A -85,B 0,C 180,E1 -764.529,E2 -764.529} C_VEL
LIN {X 0,Y 601.401,Z 340.195,A -85,B 0,C 180,E1 -766.43,E2 -766.43} C_VEL
LIN {X 0,Y 601.348,Z 340.198,A -85,B 0,C 180,E1 -769.119,E2 -769.119} C_VEL
LIN {X 0,Y 601.379,Z 340.201,A -85,B 0,C 180,E1 -771.728,E2 -771.728} C_VEL
LIN {X 0,Y 601.372,Z 340.2,A -85,B 0,C 180,E1 -774.244,E2 -774.244} C_VEL
LIN {X 0,Y 601.382,Z 340.194,A -85,B 0,C 180,E1 -776.683,E2 -776.683} C_VEL
LIN {X 0,Y 601.377,Z 340.195,A -85,B 0,C 180,E1 -779.055,E2 -779.055} C_VEL
LIN {X 0,Y 601.38,Z 340.198,A -85,B 0,C 180,E1 -781.37,E2 -781.37} C_VEL
LIN {X 0,Y 601.39,Z 340.197,A -85,B 0,C 180,E1 -784.38,E2 -784.38} C_VEL
LIN {X 0,Y 601.379,Z 340.221,A -85,B 0,C 180,E1 -784.518,E2 -784.518} C_VEL
LIN {X 0,Y 601.836,Z 343.732,A -85,B 0,C 180,E1 -784.955,E2 -784.955} C_VEL
LIN {X 0,Y 601.774,Z 366.068,A -85,B 0,C 180,E1 -787.568,E2 -787.568} C_VEL
LIN {X 0,Y 601.684,Z 390.551,A -85,B 0,C 180,E1 -790.377,E2 -790.377} C_VEL
LIN {X 0,Y 601.631,Z 398.864,A -85,B 0,C 180,E1 -791.319,E2 -791.319} C_VEL
LIN {X 0,Y 602.035,Z 402.969,A -85,B 0,C 180,E1 -791.388,E2 -791.388} C_VEL
LIN {X 0,Y 601.887,Z 564.268,A -85,B 0,C 180,E1 -793.377,E2 -793.377} C_VEL
LIN {X 0,Y 601.86,Z 579.855,A -85,B 0,C 180,E1 -793.703,E2 -793.703} C_VEL
LIN {X 0,Y 601.786,Z 594.767,A -85,B 0,C 180,E1 -794.157,E2 -794.157} C_VEL
LIN {X 0,Y 601.72,Z 609.74,A -85,B 0,C 180,E1 -794.763,E2 -794.763} C_VEL
LIN {X 0,Y 601.658,Z 623.217,A -85,B 0,C 180,E1 -795.454,E2 -795.454} C_VEL
LIN {X 0,Y 601.617,Z 636.441,A -85,B 0,C 180,E1 -796.283,E2 -796.283} C_VEL
LIN {X 0,Y 601.531,Z 648.274,A -85,B 0,C 180,E1 -797.173,E2 -797.173} C_VEL
LIN {X 0,Y 601.489,Z 659.739,A -85,B 0,C 180,E1 -798.2,E2 -798.2} C_VEL
LIN {X 0,Y 601.43,Z 669.381,A -85,B 0,C 180,E1 -799.223,E2 -799.223} C_VEL
LIN {X 0,Y 601.428,Z 678.848,A -85,B 0,C 180,E1 -800.414,E2 -800.414} C_VEL
LIN {X 0,Y 601.369,Z 686.725,A -85,B 0,C 180,E1 -801.599,E2 -801.599} C_VEL
LIN {X 0,Y 601.368,Z 694.083,A -85,B 0,C 180,E1 -802.951,E2 -802.951} C_VEL
LIN {X 0,Y 601.373,Z 699.92,A -85,B 0,C 180,E1 -804.298,E2 -804.298} C_VEL
LIN {X 0,Y 601.33,Z 703.38,A -85,B 0,C 180,E1 -805.306,E2 -805.306} C_VEL
LIN {X 0,Y 601.338,Z 706.884,A -85,B 0,C 180,E1 -806.649,E2 -806.649} C_VEL
LIN {X 0,Y 601.342,Z 709.191,A -85,B 0,C 180,E1 -807.99,E2 -807.99} C_VEL
LIN {X 0,Y 601.335,Z 710.35,A -85,B 0,C 180,E1 -809.329,E2 -809.329} C_VEL
LIN {X 0,Y 601.335,Z 710.35,A -85,B 0,C 180,E1 -810.669,E2 -810.669} C_VEL
LIN {X 0,Y 601.342,Z 709.193,A -85,B 0,C 180,E1 -812.008,E2 -812.008} C_VEL
LIN {X 0,Y 601.337,Z 706.888,A -85,B 0,C 180,E1 -813.349,E2 -813.349} C_VEL
LIN {X 0,Y 601.329,Z 703.386,A -85,B 0,C 180,E1 -814.692,E2 -814.692} C_VEL
LIN {X 0,Y 601.356,Z 698.612,A -85,B 0,C 180,E1 -816.037,E2 -816.037} C_VEL
LIN {X 0,Y 601.365,Z 692.431,A -85,B 0,C 180,E1 -817.385,E2 -817.385} C_VEL
LIN {X 0,Y 601.386,Z 684.66,A -85,B 0,C 180,E1 -818.737,E2 -818.737} C_VEL
LIN {X 0,Y 601.428,Z 676.379,A -85,B 0,C 180,E1 -819.924,E2 -819.924} C_VEL
LIN {X 0,Y 601.459,Z 665.939,A -85,B 0,C 180,E1 -821.164,E2 -821.164} C_VEL
LIN {X 0,Y 601.514,Z 656.204,A -85,B 0,C 180,E1 -822.139,E2 -822.139} C_VEL
LIN {X 0,Y 601.57,Z 644.031,A -85,B 0,C 180,E1 -823.167,E2 -823.167} C_VEL
LIN {X 0,Y 601.603,Z 632.095,A -85,B 0,C 180,E1 -824.01,E2 -824.01} C_VEL
LIN {X 0,Y 601.661,Z 618.549,A -85,B 0,C 180,E1 -824.803,E2 -824.803} C_VEL
LIN {X 0,Y 601.762,Z 603.87,A -85,B 0,C 180,E1 -825.494,E2 -825.494} C_VEL
LIN {X 0,Y 601.785,Z 589.654,A -85,B 0,C 180,E1 -826.015,E2 -826.015} C_VEL
LIN {X 0,Y 601.853,Z 574.746,A -85,B 0,C 180,E1 -826.419,E2 -826.419} C_VEL
LIN {X 0,Y 601.864,Z 559.799,A -85,B 0,C 180,E1 -826.689,E2 -826.689} C_VEL
LIN {X 0,Y 601.906,Z 400.484,A -85,B 0,C 180,E1 -828.647,E2 -828.647} C_VEL
LIN {X 0,Y 601.651,Z 398.747,A -85,B 0,C 180,E1 -828.694,E2 -828.694} C_VEL
LIN {X 0,Y 601.745,Z 373.403,A -85,B 0,C 180,E1 -831.585,E2 -831.585} C_VEL
LIN {X 0,Y 601.874,Z 349.312,A -85,B 0,C 180,E1 -834.385,E2 -834.385} C_VEL
LIN {X 0,Y 601.808,Z 342.19,A -85,B 0,C 180,E1 -835.229,E2 -835.229} C_VEL
LIN {X 0,Y 601.399,Z 340.197,A -85,B 0,C 180,E1 -835.502,E2 -835.502} C_VEL
LIN {X 0,Y 601.403,Z 340.195,A -85,B 0,C 180,E1 -838.627,E2 -838.627} C_VEL
LIN {X 0,Y 601.392,Z 340.193,A -85,B 0,C 180,E1 -840.942,E2 -840.942} C_VEL
LIN {X 0,Y 601.397,Z 340.191,A -85,B 0,C 180,E1 -843.314,E2 -843.314} C_VEL
LIN {X 0,Y 601.383,Z 340.203,A -85,B 0,C 180,E1 -846.258,E2 -846.258} C_VEL
LIN {X 0,Y 601.37,Z 340.195,A -85,B 0,C 180,E1 -849.128,E2 -849.128} C_VEL
LIN {X 0,Y 601.412,Z 340.193,A -85,B 0,C 180,E1 -851.764,E2 -851.764} C_VEL
LIN {X 0,Y 601.386,Z 340.197,A -85,B 0,C 180,E1 -854.532,E2 -854.532} C_VEL
LIN {X 0,Y 601.359,Z 340.196,A -85,B 0,C 180,E1 -857.413,E2 -857.413} C_VEL
LIN {X 0,Y 601.386,Z 340.2,A -85,B 0,C 180,E1 -860.003,E2 -860.003} C_VEL
LIN {X 0,Y 601.383,Z 340.196,A -85,B 0,C 180,E1 -862.622,E2 -862.622} C_VEL
LIN {X 0,Y 601.358,Z 340.196,A -85,B 0,C 180,E1 -865.064,E2 -865.064} C_VEL
LIN {X 0,Y 601.391,Z 340.193,A -85,B 0,C 180,E1 -867.482,E2 -867.482} C_VEL
LIN {X 0,Y 601.414,Z 340.195,A -85,B 0,C 180,E1 -869.851,E2 -869.851} C_VEL
LIN {X 0,Y 601.364,Z 340.196,A -85,B 0,C 180,E1 -872.885,E2 -872.885} C_VEL
LIN {X 0,Y 601.424,Z 340.194,A -85,B 0,C 180,E1 -875.858,E2 -875.858} C_VEL
LIN {X 0,Y 601.369,Z 340.196,A -85,B 0,C 180,E1 -878.759,E2 -878.759} C_VEL
LIN {X 0,Y 601.386,Z 340.195,A -85,B 0,C 180,E1 -881.607,E2 -881.607} C_VEL
LIN {X 0,Y 601.376,Z 340.199,A -85,B 0,C 180,E1 -884.408,E2 -884.408} C_VEL
LIN {X 0,Y 601.378,Z 340.197,A -85,B 0,C 180,E1 -886.483,E2 -886.483} C_VEL
LIN {X 0,Y 601.348,Z 340.197,A -85,B 0,C 180,E1 -889.223,E2 -889.223} C_VEL
LIN {X 0,Y 601.42,Z 340.197,A -85,B 0,C 180,E1 -891.939,E2 -891.939} C_VEL
LIN {X 0,Y 601.377,Z 340.195,A -85,B 0,C 180,E1 -894.636,E2 -894.636} C_VEL
LIN {X 0,Y 601.384,Z 340.194,A -85,B 0,C 180,E1 -897.321,E2 -897.321} C_VEL
LIN {X 0,Y 601.431,Z 340.198,A -85,B 0,C 180,E1 -900,E2 -900} C_VEL
LIN {X 0,Y 601.383,Z 340.194,A -85,B 0,C 180,E1 -902.679,E2 -902.679} C_VEL
LIN {X 0,Y 601.374,Z 340.196,A -85,B 0,C 180,E1 -905.365,E2 -905.365} C_VEL
LIN {X 0,Y 601.419,Z 340.198,A -85,B 0,C 180,E1 -908.061,E2 -908.061} C_VEL
LIN {X 0,Y 601.364,Z 340.195,A -85,B 0,C 180,E1 -910.99,E2 -910.99} C_VEL
LIN {X 0,Y 601.366,Z 340.199,A -85,B 0,C 180,E1 -912.341,E2 -912.341} C_VEL
LIN {X 0,Y 600.673,Z 340.284,A -85,B 0,C 180,E1 -912.9,E2 -912.9} C_VEL
LIN {X 0,Y 597.816,Z 340.645,A -85,B 0,C 180,E1 -913.809,E2 -913.809} C_VEL
LIN {X 0,Y 595.42,Z 340.939,A -85,B 0,C 180,E1 -914.539,E2 -914.539} C_VEL
LIN {X 0,Y 594.395,Z 341.064,A -85,B 0,C 180,E1 -915.103,E2 -915.103} C_VEL
LIN {X 0,Y 594.312,Z 341.075,A -85,B 0,C 180,E1 -915.293,E2 -915.293} C_VEL
LIN {X 0,Y 594.324,Z 341.083,A -85,B 0,C 180,E1 -917.906,E2 -917.906} C_VEL
LIN {X 0,Y 594.363,Z 341.068,A -85,B 0,C 180,E1 -920.777,E2 -920.777} C_VEL
LIN {X 0,Y 594.347,Z 341.076,A -85,B 0,C 180,E1 -923.706,E2 -923.706} C_VEL
LIN {X 0,Y 594.328,Z 341.072,A -85,B 0,C 180,E1 -926.703,E2 -926.703} C_VEL
LIN {X 0,Y 594.323,Z 341.072,A -85,B 0,C 180,E1 -929.002,E2 -929.002} C_VEL
LIN {X 0,Y 594.356,Z 341.074,A -85,B 0,C 180,E1 -931.642,E2 -931.642} C_VEL
LIN {X 0,Y 594.344,Z 341.071,A -85,B 0,C 180,E1 -934.583,E2 -934.583} C_VEL
LIN {X 0,Y 594.351,Z 341.075,A -85,B 0,C 180,E1 -937.606,E2 -937.606} C_VEL
LIN {X 0,Y 594.342,Z 341.071,A -85,B 0,C 180,E1 -940.57,E2 -940.57} C_VEL
LIN {X 0,Y 594.33,Z 341.074,A -85,B 0,C 180,E1 -943.303,E2 -943.303} C_VEL
LIN {X 0,Y 594.335,Z 341.076,A -85,B 0,C 180,E1 -946.164,E2 -946.164} C_VEL
LIN {X 0,Y 594.356,Z 341.069,A -85,B 0,C 180,E1 -948.536,E2 -948.536} C_VEL
LIN {X 0,Y 594.357,Z 341.071,A -85,B 0,C 180,E1 -951.299,E2 -951.299} C_VEL
LIN {X 0,Y 594.338,Z 341.081,A -85,B 0,C 180,E1 -953.756,E2 -953.756} C_VEL
LIN {X 0,Y 594.354,Z 341.072,A -85,B 0,C 180,E1 -956.239,E2 -956.239} C_VEL
LIN {X 0,Y 594.353,Z 341.069,A -85,B 0,C 180,E1 -958.65,E2 -958.65} C_VEL
LIN {X 0,Y 594.334,Z 341.072,A -85,B 0,C 180,E1 -961.051,E2 -961.051} C_VEL
LIN {X 0,Y 594.353,Z 341.074,A -85,B 0,C 180,E1 -964.056,E2 -964.056} C_VEL
LIN {X 0,Y 594.366,Z 341.069,A -85,B 0,C 180,E1 -966.296,E2 -966.296} C_VEL
LIN {X 0,Y 594.385,Z 341.067,A -85,B 0,C 180,E1 -969.225,E2 -969.225} C_VEL
LIN {X 0,Y 594.334,Z 341.075,A -85,B 0,C 180,E1 -972.096,E2 -972.096} C_VEL
LIN {X 0,Y 594.342,Z 341.073,A -85,B 0,C 180,E1 -974.22,E2 -974.22} C_VEL
LIN {X 0,Y 594.364,Z 341.069,A -85,B 0,C 180,E1 -976.322,E2 -976.322} C_VEL
LIN {X 0,Y 594.364,Z 341.069,A -85,B 0,C 180,E1 -979.096,E2 -979.096} C_VEL
LIN {X 0,Y 594.379,Z 341.073,A -85,B 0,C 180,E1 -981.844,E2 -981.844} C_VEL
LIN {X 0,Y 594.361,Z 341.068,A -85,B 0,C 180,E1 -984.573,E2 -984.573} C_VEL
LIN {X 0,Y 594.386,Z 341.069,A -85,B 0,C 180,E1 -987.29,E2 -987.29} C_VEL
LIN {X 0,Y 594.414,Z 341.066,A -85,B 0,C 180,E1 -990.001,E2 -990.001} C_VEL
LIN {X 0,Y 594.374,Z 341.066,A -85,B 0,C 180,E1 -992.712,E2 -992.712} C_VEL
LIN {X 0,Y 594.375,Z 341.073,A -85,B 0,C 180,E1 -995.429,E2 -995.429} C_VEL
LIN {X 0,Y 594.382,Z 341.067,A -85,B 0,C 180,E1 -998.158,E2 -998.158} C_VEL
LIN {X 0,Y 594.369,Z 341.069,A -85,B 0,C 180,E1 -1001.061,E2 -1001.061} C_VEL
LIN {X 0,Y 594.375,Z 341.075,A -85,B 0,C 180,E1 -1003.68,E2 -1003.68} C_VEL
LIN {X 0,Y 594.337,Z 341.071,A -85,B 0,C 180,E1 -1006.699,E2 -1006.699} C_VEL
LIN {X 0,Y 594.362,Z 341.074,A -85,B 0,C 180,E1 -1009.335,E2 -1009.335} C_VEL
LIN {X 0,Y 594.357,Z 341.078,A -85,B 0,C 180,E1 -1011.504,E2 -1011.504} C_VEL
LIN {X 0,Y 594.372,Z 341.066,A -85,B 0,C 180,E1 -1014.448,E2 -1014.448} C_VEL
LIN {X 0,Y 594.36,Z 341.068,A -85,B 0,C 180,E1 -1016.702,E2 -1016.702} C_VEL
LIN {X 0,Y 594.376,Z 341.068,A -85,B 0,C 180,E1 -1019,E2 -1019} C_VEL
LIN {X 0,Y 594.377,Z 341.074,A -85,B 0,C 180,E1 -1021.642,E2 -1021.642} C_VEL
LIN {X 0,Y 594.377,Z 341.067,A -85,B 0,C 180,E1 -1024.137,E2 -1024.137} C_VEL
LIN {X 0,Y 594.378,Z 341.07,A -85,B 0,C 180,E1 -1027.088,E2 -1027.088} C_VEL
LIN {X 0,Y 594.358,Z 341.074,A -85,B 0,C 180,E1 -1029.772,E2 -1029.772} C_VEL
LIN {X 0,Y 594.346,Z 341.07,A -85,B 0,C 180,E1 -1032.378,E2 -1032.378} C_VEL
LIN {X 0,Y 594.342,Z 341.072,A -85,B 0,C 180,E1 -1034.806,E2 -1034.806} C_VEL
LIN {X 0,Y 594.37,Z 341.076,A -85,B 0,C 180,E1 -1037.624,E2 -1037.624} C_VEL
LIN {X 0,Y 594.398,Z 341.121,A -85,B 0,C 180,E1 -1038.277,E2 -1038.277} C_VEL
LIN {X 0,Y 594.742,Z 345.555,A -85,B 0,C 180,E1 -1038.892,E2 -1038.892} C_VEL
LIN {X 0,Y 594.678,Z 364.687,A -85,B 0,C 180,E1 -1041.458,E2 -1041.458} C_VEL
LIN {X 0,Y 594.638,Z 369.89,A -85,B 0,C 180,E1 -1042.148,E2 -1042.148} C_VEL
LIN {X 0,Y 595.257,Z 373.271,A -85,B 0,C 180,E1 -1042.217,E2 -1042.217} C_VEL
LIN {X 0,Y 595.113,Z 534.336,A -85,B 0,C 180,E1 -1044.227,E2 -1044.227} C_VEL
LIN {X 0,Y 595.009,Z 550.067,A -85,B 0,C 180,E1 -1044.561,E2 -1044.561} C_VEL
LIN {X 0,Y 594.914,Z 565.603,A -85,B 0,C 180,E1 -1045.043,E2 -1045.043} C_VEL
LIN {X 0,Y 594.825,Z 579.83,A -85,B 0,C 180,E1 -1045.633,E2 -1045.633} C_VEL
LIN {X 0,Y 594.723,Z 593.841,A -85,B 0,C 180,E1 -1046.362,E2 -1046.362} C_VEL
LIN {X 0,Y 594.646,Z 606.937,A -85,B 0,C 180,E1 -1047.197,E2 -1047.197} C_VEL
LIN {X 0,Y 594.562,Z 619.479,A -85,B 0,C 180,E1 -1048.164,E2 -1048.164} C_VEL
LIN {X 0,Y 594.454,Z 631.212,A -85,B 0,C 180,E1 -1049.247,E2 -1049.247} C_VEL
LIN {X 0,Y 594.401,Z 641.776,A -85,B 0,C 180,E1 -1050.42,E2 -1050.42} C_VEL
LIN {X 0,Y 594.347,Z 650.547,A -85,B 0,C 180,E1 -1051.579,E2 -1051.579} C_VEL
LIN {X 0,Y 594.299,Z 658.923,A -85,B 0,C 180,E1 -1052.916,E2 -1052.916} C_VEL
LIN {X 0,Y 594.281,Z 664.752,A -85,B 0,C 180,E1 -1054.051,E2 -1054.051} C_VEL
LIN {X 0,Y 594.264,Z 669.563,A -85,B 0,C 180,E1 -1055.175,E2 -1055.175} C_VEL
LIN {X 0,Y 594.232,Z 674.456,A -85,B 0,C 180,E1 -1056.659,E2 -1056.659} C_VEL
LIN {X 0,Y 594.256,Z 677.113,A -85,B 0,C 180,E1 -1057.762,E2 -1057.762} C_VEL
LIN {X 0,Y 594.253,Z 679.436,A -85,B 0,C 180,E1 -1059.219,E2 -1059.219} C_VEL
LIN {X 0,Y 594.211,Z 680.418,A -85,B 0,C 180,E1 -1060.66,E2 -1060.66} C_VEL
LIN {X 0,Y 594.205,Z 680.131,A -85,B 0,C 180,E1 -1062.09,E2 -1062.09} C_VEL
LIN {X 0,Y 594.242,Z 678.591,A -85,B 0,C 180,E1 -1063.51,E2 -1063.51} C_VEL
LIN {X 0,Y 594.226,Z 675.797,A -85,B 0,C 180,E1 -1064.918,E2 -1064.918} C_VEL
LIN {X 0,Y 594.257,Z 671.729,A -85,B 0,C 180,E1 -1066.318,E2 -1066.318} C_VEL
LIN {X 0,Y 594.28,Z 666.283,A -85,B 0,C 180,E1 -1067.709,E2 -1067.709} C_VEL
LIN {X 0,Y 594.319,Z 659.378,A -85,B 0,C 180,E1 -1069.093,E2 -1069.093} C_VEL
LIN {X 0,Y 594.332,Z 650.826,A -85,B 0,C 180,E1 -1070.471,E2 -1070.471} C_VEL
LIN {X 0,Y 594.407,Z 641.761,A -85,B 0,C 180,E1 -1071.672,E2 -1071.672} C_VEL
LIN {X 0,Y 594.449,Z 630.95,A -85,B 0,C 180,E1 -1072.869,E2 -1072.869} C_VEL
LIN {X 0,Y 594.556,Z 618.857,A -85,B 0,C 180,E1 -1073.978,E2 -1073.978} C_VEL
LIN {X 0,Y 594.656,Z 605.371,A -85,B 0,C 180,E1 -1074.999,E2 -1074.999} C_VEL
LIN {X 0,Y 594.765,Z 591.696,A -85,B 0,C 180,E1 -1075.849,E2 -1075.849} C_VEL
LIN {X 0,Y 594.839,Z 578.275,A -85,B 0,C 180,E1 -1076.528,E2 -1076.528} C_VEL
LIN {X 0,Y 594.929,Z 563.424,A -85,B 0,C 180,E1 -1077.122,E2 -1077.122} C_VEL
LIN {X 0,Y 595.044,Z 547.628,A -85,B 0,C 180,E1 -1077.588,E2 -1077.588} C_VEL
LIN {X 0,Y 595.092,Z 532.876,A -85,B 0,C 180,E1 -1077.885,E2 -1077.885} C_VEL
LIN {X 0,Y 595.271,Z 373.247,A -85,B 0,C 180,E1 -1079.873,E2 -1079.873} C_VEL
LIN {X 0,Y 594.645,Z 369.773,A -85,B 0,C 180,E1 -1079.957,E2 -1079.957} C_VEL
LIN {X 0,Y 594.758,Z 349.165,A -85,B 0,C 180,E1 -1082.709,E2 -1082.709} C_VEL
LIN {X 0,Y 594.72,Z 342.912,A -85,B 0,C 180,E1 -1083.557,E2 -1083.557} C_VEL
LIN {X 0,Y 594.368,Z 341.073,A -85,B 0,C 180,E1 -1083.856,E2 -1083.856} C_VEL
LIN {X 0,Y 594.388,Z 341.072,A -85,B 0,C 180,E1 -1086.79,E2 -1086.79} C_VEL
LIN {X 0,Y 594.35,Z 341.07,A -85,B 0,C 180,E1 -1089.529,E2 -1089.529} C_VEL
LIN {X 0,Y 594.388,Z 341.072,A -85,B 0,C 180,E1 -1092.288,E2 -1092.288} C_VEL
LIN {X 0,Y 594.362,Z 341.07,A -85,B 0,C 180,E1 -1095.078,E2 -1095.078} C_VEL
LIN {X 0,Y 594.371,Z 341.068,A -85,B 0,C 180,E1 -1097.194,E2 -1097.194} C_VEL
LIN {X 0,Y 594.365,Z 341.073,A -85,B 0,C 180,E1 -1100.054,E2 -1100.054} C_VEL
LIN {X 0,Y 594.352,Z 341.071,A -85,B 0,C 180,E1 -1102.968,E2 -1102.968} C_VEL
LIN {X 0,Y 594.327,Z 341.072,A -85,B 0,C 180,E1 -1105.195,E2 -1105.195} C_VEL
LIN {X 0,Y 594.345,Z 341.071,A -85,B 0,C 180,E1 -1107.518,E2 -1107.518} C_VEL
LIN {X 0,Y 594.364,Z 341.073,A -85,B 0,C 180,E1 -1110.56,E2 -1110.56} C_VEL
LIN {X 0,Y 594.341,Z 341.071,A -85,B 0,C 180,E1 -1112.952,E2 -1112.952} C_VEL
LIN {X 0,Y 594.31,Z 341.075,A -85,B 0,C 180,E1 -1115.412,E2 -1115.412} C_VEL
LIN {X 0,Y 594.365,Z 341.075,A -85,B 0,C 180,E1 -1117.942,E2 -1117.942} C_VEL
LIN {X 0,Y 594.324,Z 341.073,A -85,B 0,C 180,E1 -1120.815,E2 -1120.815} C_VEL
LIN {X 0,Y 594.336,Z 341.072,A -85,B 0,C 180,E1 -1123.302,E2 -1123.302} C_VEL
LIN {X 0,Y 594.334,Z 341.079,A -85,B 0,C 180,E1 -1126.164,E2 -1126.164} C_VEL
LIN {X 0,Y 594.349,Z 341.072,A -85,B 0,C 180,E1 -1128.533,E2 -1128.533} C_VEL
LIN {X 0,Y 594.326,Z 341.074,A -85,B 0,C 180,E1 -1131.303,E2 -1131.303} C_VEL
LIN {X 0,Y 594.339,Z 341.079,A -85,B 0,C 180,E1 -1133.754,E2 -1133.754} C_VEL
LIN {X 0,Y 594.344,Z 341.075,A -85,B 0,C 180,E1 -1136.236,E2 -1136.236} C_VEL
LIN {X 0,Y 594.325,Z 341.074,A -85,B 0,C 180,E1 -1138.646,E2 -1138.646} C_VEL
LIN {X 0,Y 594.338,Z 341.073,A -85,B 0,C 180,E1 -1141.05,E2 -1141.05} C_VEL
LIN {X 0,Y 594.351,Z 341.078,A -85,B 0,C 180,E1 -1143.984,E2 -1143.984} C_VEL
LIN {X 0,Y 594.363,Z 341.196,A -85,B 0,C 180,E1 -1144.313,E2 -1144.313} C_VEL
LIN {X 0,Y 595.047,Z 345.293,A -85,B 0,C 180,E1 -1144.837,E2 -1144.837} C_VEL
LIN {X 0,Y 594.912,Z 368.935,A -85,B 0,C 180,E1 -1147.632,E2 -1147.632} C_VEL
LIN {X 0,Y 594.759,Z 393.673,A -85,B 0,C 180,E1 -1150.499,E2 -1150.499} C_VEL
LIN {X 0,Y 594.703,Z 398.88,A -85,B 0,C 180,E1 -1151.095,E2 -1151.095} C_VEL
LIN {X 0,Y 595.319,Z 402.4,A -85,B 0,C 180,E1 -1151.163,E2 -1151.163} C_VEL
LIN {X 0,Y 595.082,Z 565.361,A -85,B 0,C 180,E1 -1153.199,E2 -1153.199} C_VEL
LIN {X 0,Y 595.014,Z 580.678,A -85,B 0,C 180,E1 -1153.531,E2 -1153.531} C_VEL
LIN {X 0,Y 594.934,Z 596.024,A -85,B 0,C 180,E1 -1154.014,E2 -1154.014} C_VEL
LIN {X 0,Y 594.858,Z 609.743,A -85,B 0,C 180,E1 -1154.583,E2 -1154.583} C_VEL
LIN {X 0,Y 594.733,Z 623.22,A -85,B 0,C 180,E1 -1155.281,E2 -1155.281} C_VEL
LIN {X 0,Y 594.682,Z 635.779,A -85,B 0,C 180,E1 -1156.074,E2 -1156.074} C_VEL
LIN {X 0,Y 594.56,Z 648.275,A -85,B 0,C 180,E1 -1157.02,E2 -1157.02} C_VEL
LIN {X 0,Y 594.467,Z 659.739,A -85,B 0,C 180,E1 -1158.059,E2 -1158.059} C_VEL
LIN {X 0,Y 594.388,Z 669.382,A -85,B 0,C 180,E1 -1159.094,E2 -1159.094} C_VEL
LIN {X 0,Y 594.367,Z 678.849,A -85,B 0,C 180,E1 -1160.299,E2 -1160.299} C_VEL
LIN {X 0,Y 594.311,Z 686.725,A -85,B 0,C 180,E1 -1161.499,E2 -1161.499} C_VEL
LIN {X 0,Y 594.292,Z 694.084,A -85,B 0,C 180,E1 -1162.866,E2 -1162.866} C_VEL
LIN {X 0,Y 594.298,Z 699.921,A -85,B 0,C 180,E1 -1164.23,E2 -1164.23} C_VEL
LIN {X 0,Y 594.232,Z 703.381,A -85,B 0,C 180,E1 -1165.25,E2 -1165.25} C_VEL
LIN {X 0,Y 594.257,Z 706.885,A -85,B 0,C 180,E1 -1166.609,E2 -1166.609} C_VEL
LIN {X 0,Y 594.241,Z 709.192,A -85,B 0,C 180,E1 -1167.966,E2 -1167.966} C_VEL
LIN {X 0,Y 594.235,Z 710.35,A -85,B 0,C 180,E1 -1169.321,E2 -1169.321} C_VEL
LIN {X 0,Y 594.235,Z 710.35,A -85,B 0,C 180,E1 -1170.677,E2 -1170.677} C_VEL
LIN {X 0,Y 594.241,Z 709.193,A -85,B 0,C 180,E1 -1172.032,E2 -1172.032} C_VEL
LIN {X 0,Y 594.257,Z 706.888,A -85,B 0,C 180,E1 -1173.389,E2 -1173.389} C_VEL
LIN {X 0,Y 594.232,Z 703.387,A -85,B 0,C 180,E1 -1174.748,E2 -1174.748} C_VEL
LIN {X 0,Y 594.277,Z 698.612,A -85,B 0,C 180,E1 -1176.109,E2 -1176.109} C_VEL
LIN {X 0,Y 594.286,Z 692.431,A -85,B 0,C 180,E1 -1177.473,E2 -1177.473} C_VEL
LIN {X 0,Y 594.329,Z 684.659,A -85,B 0,C 180,E1 -1178.842,E2 -1178.842} C_VEL
LIN {X 0,Y 594.387,Z 676.379,A -85,B 0,C 180,E1 -1180.043,E2 -1180.043} C_VEL
LIN {X 0,Y 594.432,Z 666.565,A -85,B 0,C 180,E1 -1181.23,E2 -1181.23} C_VEL
LIN {X 0,Y 594.53,Z 656.204,A -85,B 0,C 180,E1 -1182.284,E2 -1182.284} C_VEL
LIN {X 0,Y 594.581,Z 644.032,A -85,B 0,C 180,E1 -1183.325,E2 -1183.325} C_VEL
LIN {X 0,Y 594.691,Z 632.092,A -85,B 0,C 180,E1 -1184.177,E2 -1184.177} C_VEL
LIN {X 0,Y 594.779,Z 618.546,A -85,B 0,C 180,E1 -1184.979,E2 -1184.979} C_VEL
LIN {X 0,Y 594.902,Z 603.868,A -85,B 0,C 180,E1 -1185.677,E2 -1185.677} C_VEL
LIN {X 0,Y 594.966,Z 589.654,A -85,B 0,C 180,E1 -1186.203,E2 -1186.203} C_VEL
LIN {X 0,Y 595.042,Z 575.171,A -85,B 0,C 180,E1 -1186.602,E2 -1186.602} C_VEL
LIN {X 0,Y 595.064,Z 559.799,A -85,B 0,C 180,E1 -1186.885,E2 -1186.885} C_VEL
LIN {X 0,Y 595.216,Z 401.589,A -85,B 0,C 180,E1 -1188.85,E2 -1188.85} C_VEL
LIN {X 0,Y 594.73,Z 398.808,A -85,B 0,C 180,E1 -1188.913,E2 -1188.913} C_VEL
LIN {X 0,Y 594.892,Z 373.403,A -85,B 0,C 180,E1 -1191.846,E2 -1191.846} C_VEL
LIN {X 0,Y 595.042,Z 350.246,A -85,B 0,C 180,E1 -1194.572,E2 -1194.572} C_VEL
LIN {X 0,Y 594.954,Z 343.751,A -85,B 0,C 180,E1 -1195.353,E2 -1195.353} C_VEL
LIN {X 0,Y 594.354,Z 341.077,A -85,B 0,C 180,E1 -1195.708,E2 -1195.708} C_VEL
LIN {X 0,Y 594.355,Z 341.079,A -85,B 0,C 180,E1 -1198.227,E2 -1198.227} C_VEL
LIN {X 0,Y 594.368,Z 341.073,A -85,B 0,C 180,E1 -1200.559,E2 -1200.559} C_VEL
LIN {X 0,Y 594.364,Z 341.068,A -85,B 0,C 180,E1 -1202.949,E2 -1202.949} C_VEL
LIN {X 0,Y 594.309,Z 341.075,A -85,B 0,C 180,E1 -1205.41,E2 -1205.41} C_VEL
LIN {X 0,Y 594.364,Z 341.073,A -85,B 0,C 180,E1 -1207.941,E2 -1207.941} C_VEL
LIN {X 0,Y 594.348,Z 341.071,A -85,B 0,C 180,E1 -1210.819,E2 -1210.819} C_VEL
LIN {X 0,Y 594.331,Z 341.071,A -85,B 0,C 180,E1 -1213.301,E2 -1213.301} C_VEL
LIN {X 0,Y 594.333,Z 341.082,A -85,B 0,C 180,E1 -1216.162,E2 -1216.162} C_VEL
LIN {X 0,Y 594.355,Z 341.073,A -85,B 0,C 180,E1 -1218.534,E2 -1218.534} C_VEL
LIN {X 0,Y 594.351,Z 341.069,A -85,B 0,C 180,E1 -1221.297,E2 -1221.297} C_VEL
LIN {X 0,Y 594.332,Z 341.075,A -85,B 0,C 180,E1 -1223.754,E2 -1223.754} C_VEL
LIN {X 0,Y 594.356,Z 341.077,A -85,B 0,C 180,E1 -1226.237,E2 -1226.237} C_VEL
LIN {X 0,Y 594.344,Z 341.072,A -85,B 0,C 180,E1 -1228.648,E2 -1228.648} C_VEL
LIN {X 0,Y 594.322,Z 341.072,A -85,B 0,C 180,E1 -1231.05,E2 -1231.05} C_VEL
LIN {X 0,Y 594.348,Z 341.079,A -85,B 0,C 180,E1 -1234.055,E2 -1234.055} C_VEL
LIN {X 0,Y 594.347,Z 341.076,A -85,B 0,C 180,E1 -1236.294,E2 -1236.294} C_VEL
LIN {X 0,Y 594.363,Z 341.067,A -85,B 0,C 180,E1 -1239.223,E2 -1239.223} C_VEL
LIN {X 0,Y 594.324,Z 341.083,A -85,B 0,C 180,E1 -1242.094,E2 -1242.094} C_VEL
LIN {X 0,Y 594.329,Z 341.08,A -85,B 0,C 180,E1 -1244.218,E2 -1244.218} C_VEL
LIN {X 0,Y 594.35,Z 341.075,A -85,B 0,C 180,E1 -1246.32,E2 -1246.32} C_VEL
LIN {X 0,Y 594.326,Z 341.072,A -85,B 0,C 180,E1 -1249.094,E2 -1249.094} C_VEL
LIN {X 0,Y 594.362,Z 341.075,A -85,B 0,C 180,E1 -1251.843,E2 -1251.843} C_VEL
LIN {X 0,Y 594.349,Z 341.071,A -85,B 0,C 180,E1 -1254.572,E2 -1254.572} C_VEL
LIN {X 0,Y 594.352,Z 341.069,A -85,B 0,C 180,E1 -1257.289,E2 -1257.289} C_VEL
LIN {X 0,Y 594.399,Z 341.074,A -85,B 0,C 180,E1 -1260,E2 -1260} C_VEL
LIN {X 0,Y 594.351,Z 341.07,A -85,B 0,C 180,E1 -1262.711,E2 -1262.711} C_VEL
LIN {X 0,Y 594.343,Z 341.072,A -85,B 0,C 180,E1 -1265.428,E2 -1265.428} C_VEL
LIN {X 0,Y 594.361,Z 341.075,A -85,B 0,C 180,E1 -1268.158,E2 -1268.158} C_VEL
LIN {X 0,Y 594.329,Z 341.072,A -85,B 0,C 180,E1 -1271.052,E2 -1271.052} C_VEL
LIN {X 0,Y 594.35,Z 341.075,A -85,B 0,C 180,E1 -1273.68,E2 -1273.68} C_VEL
LIN {X 0,Y 594.312,Z 341.075,A -85,B 0,C 180,E1 -1275.293,E2 -1275.293} C_VEL
LIN {X 0,Y 593.647,Z 341.166,A -85,B 0,C 180,E1 -1275.859,E2 -1275.859} C_VEL
LIN {X 0,Y 590.791,Z 341.525,A -85,B 0,C 180,E1 -1276.777,E2 -1276.777} C_VEL
LIN {X 0,Y 588.382,Z 341.824,A -85,B 0,C 180,E1 -1277.515,E2 -1277.515} C_VEL
LIN {X 0,Y 587.354,Z 341.948,A -85,B 0,C 180,E1 -1278.085,E2 -1278.085} C_VEL
LIN {X 0,Y 587.275,Z 341.955,A -85,B 0,C 180,E1 -1278.278,E2 -1278.278} C_VEL
LIN {X 0,Y 587.3,Z 341.947,A -85,B 0,C 180,E1 -1281.039,E2 -1281.039} C_VEL
LIN {X 0,Y 587.29,Z 341.957,A -85,B 0,C 180,E1 -1284.009,E2 -1284.009} C_VEL
LIN {X 0,Y 587.28,Z 341.954,A -85,B 0,C 180,E1 -1286.282,E2 -1286.282} C_VEL
LIN {X 0,Y 587.286,Z 341.949,A -85,B 0,C 180,E1 -1289.126,E2 -1289.126} C_VEL
LIN {X 0,Y 587.327,Z 341.954,A -85,B 0,C 180,E1 -1291.836,E2 -1291.836} C_VEL
LIN {X 0,Y 587.322,Z 341.947,A -85,B 0,C 180,E1 -1294.347,E2 -1294.347} C_VEL
LIN {X 0,Y 587.306,Z 341.953,A -85,B 0,C 180,E1 -1297.611,E2 -1297.611} C_VEL
LIN {X 0,Y 587.291,Z 341.952,A -85,B 0,C 180,E1 -1300.257,E2 -1300.257} C_VEL
LIN {X 0,Y 587.274,Z 341.951,A -85,B 0,C 180,E1 -1303.116,E2 -1303.116} C_VEL
LIN {X 0,Y 587.29,Z 341.955,A -85,B 0,C 180,E1 -1306.048,E2 -1306.048} C_VEL
LIN {X 0,Y 587.298,Z 341.947,A -85,B 0,C 180,E1 -1308.842,E2 -1308.842} C_VEL
LIN {X 0,Y 587.306,Z 341.952,A -85,B 0,C 180,E1 -1311.521,E2 -1311.521} C_VEL
LIN {X 0,Y 587.27,Z 341.956,A -85,B 0,C 180,E1 -1314.1,E2 -1314.1} C_VEL
LIN {X 0,Y 587.318,Z 341.945,A -85,B 0,C 180,E1 -1316.604,E2 -1316.604} C_VEL
LIN {X 0,Y 587.326,Z 341.95,A -85,B 0,C 180,E1 -1319.493,E2 -1319.493} C_VEL
LIN {X 0,Y 587.295,Z 341.95,A -85,B 0,C 180,E1 -1322.318,E2 -1322.318} C_VEL
LIN {X 0,Y 587.305,Z 341.949,A -85,B 0,C 180,E1 -1325.241,E2 -1325.241} C_VEL
LIN {X 0,Y 587.307,Z 341.949,A -85,B 0,C 180,E1 -1328.226,E2 -1328.226} C_VEL
LIN {X 0,Y 587.328,Z 341.946,A -85,B 0,C 180,E1 -1331.152,E2 -1331.152} C_VEL
LIN {X 0,Y 587.297,Z 341.953,A -85,B 0,C 180,E1 -1334.025,E2 -1334.025} C_VEL
LIN {X 0,Y 587.348,Z 341.945,A -85,B 0,C 180,E1 -1336.155,E2 -1336.155} C_VEL
LIN {X 0,Y 587.339,Z 341.943,A -85,B 0,C 180,E1 -1338.964,E2 -1338.964} C_VEL
LIN {X 0,Y 587.338,Z 341.952,A -85,B 0,C 180,E1 -1341.745,E2 -1341.745} C_VEL
LIN {X 0,Y 587.33,Z 341.944,A -85,B 0,C 180,E1 -1344.508,E2 -1344.508} C_VEL
LIN {X 0,Y 587.352,Z 341.944,A -85,B 0,C 180,E1 -1347.258,E2 -1347.258} C_VEL
LIN {X 0,Y 587.382,Z 341.942,A -85,B 0,C 180,E1 -1350.001,E2 -1350.001} C_VEL
LIN {X 0,Y 587.343,Z 341.942,A -85,B 0,C 180,E1 -1352.744,E2 -1352.744} C_VEL
LIN {X 0,Y 587.342,Z 341.95,A -85,B 0,C 180,E1 -1355.494,E2 -1355.494} C_VEL
LIN {X 0,Y 587.34,Z 341.944,A -85,B 0,C 180,E1 -1358.257,E2 -1358.257} C_VEL
LIN {X 0,Y 587.336,Z 341.946,A -85,B 0,C 180,E1 -1361.125,E2 -1361.125} C_VEL
LIN {X 0,Y 587.333,Z 341.944,A -85,B 0,C 180,E1 -1364.246,E2 -1364.246} C_VEL
LIN {X 0,Y 587.289,Z 341.949,A -85,B 0,C 180,E1 -1366.793,E2 -1366.793} C_VEL
LIN {X 0,Y 587.308,Z 341.957,A -85,B 0,C 180,E1 -1369.577,E2 -1369.577} C_VEL
LIN {X 0,Y 587.314,Z 341.952,A -85,B 0,C 180,E1 -1371.775,E2 -1371.775} C_VEL
LIN {X 0,Y 587.317,Z 341.945,A -85,B 0,C 180,E1 -1374.761,E2 -1374.761} C_VEL
LIN {X 0,Y 587.306,Z 341.955,A -85,B 0,C 180,E1 -1377.684,E2 -1377.684} C_VEL
LIN {X 0,Y 587.321,Z 341.946,A -85,B 0,C 180,E1 -1380.172,E2 -1380.172} C_VEL
LIN {X 0,Y 587.334,Z 341.943,A -85,B 0,C 180,E1 -1382.58,E2 -1382.58} C_VEL
LIN {X 0,Y 587.307,Z 341.949,A -85,B 0,C 180,E1 -1385.058,E2 -1385.058} C_VEL
LIN {X 0,Y 587.338,Z 341.948,A -85,B 0,C 180,E1 -1387.838,E2 -1387.838} C_VEL
LIN {X 0,Y 587.309,Z 341.947,A -85,B 0,C 180,E1 -1390.256,E2 -1390.256} C_VEL
LIN {X 0,Y 587.302,Z 341.952,A -85,B 0,C 180,E1 -1393.116,E2 -1393.116} C_VEL
LIN {X 0,Y 587.304,Z 341.951,A -85,B 0,C 180,E1 -1396.047,E2 -1396.047} C_VEL
LIN {X 0,Y 587.378,Z 342.06,A -85,B 0,C 180,E1 -1398.119,E2 -1398.119} C_VEL
LIN {X 0,Y 587.857,Z 345.853,A -85,B 0,C 180,E1 -1398.66,E2 -1398.66} C_VEL
LIN {X 0,Y 587.731,Z 364.378,A -85,B 0,C 180,E1 -1401.175,E2 -1401.175} C_VEL
LIN {X 0,Y 587.685,Z 369.886,A -85,B 0,C 180,E1 -1401.915,E2 -1401.915} C_VEL
LIN {X 0,Y 588.556,Z 374.524,A -85,B 0,C 180,E1 -1402.01,E2 -1402.01} C_VEL
LIN {X 0,Y 588.301,Z 535.015,A -85,B 0,C 180,E1 -1404.039,E2 -1404.039} C_VEL
LIN {X 0,Y 588.189,Z 551.152,A -85,B 0,C 180,E1 -1404.393,E2 -1404.393} C_VEL
LIN {X 0,Y 588.062,Z 566.794,A -85,B 0,C 180,E1 -1404.896,E2 -1404.896} C_VEL
LIN {X 0,Y 587.939,Z 581.421,A -85,B 0,C 180,E1 -1405.525,E2 -1405.525} C_VEL
LIN {X 0,Y 587.808,Z 594.477,A -85,B 0,C 180,E1 -1406.222,E2 -1406.222} C_VEL
LIN {X 0,Y 587.694,Z 607.459,A -85,B 0,C 180,E1 -1407.066,E2 -1407.066} C_VEL
LIN {X 0,Y 587.582,Z 619.747,A -85,B 0,C 180,E1 -1408.032,E2 -1408.032} C_VEL
LIN {X 0,Y 587.465,Z 630.569,A -85,B 0,C 180,E1 -1409.041,E2 -1409.041} C_VEL
LIN {X 0,Y 587.367,Z 641.24,A -85,B 0,C 180,E1 -1410.227,E2 -1410.227} C_VEL
LIN {X 0,Y 587.292,Z 650.107,A -85,B 0,C 180,E1 -1411.401,E2 -1411.401} C_VEL
LIN {X 0,Y 587.228,Z 657.863,A -85,B 0,C 180,E1 -1412.636,E2 -1412.636} C_VEL
LIN {X 0,Y 587.223,Z 664.196,A -85,B 0,C 180,E1 -1413.847,E2 -1413.847} C_VEL
LIN {X 0,Y 587.182,Z 670.034,A -85,B 0,C 180,E1 -1415.234,E2 -1415.234} C_VEL
LIN {X 0,Y 587.135,Z 674.784,A -85,B 0,C 180,E1 -1416.733,E2 -1416.733} C_VEL
LIN {X 0,Y 587.146,Z 678.059,A -85,B 0,C 180,E1 -1418.219,E2 -1418.219} C_VEL
LIN {X 0,Y 587.12,Z 679.927,A -85,B 0,C 180,E1 -1419.687,E2 -1419.687} C_VEL
LIN {X 0,Y 587.158,Z 680.484,A -85,B 0,C 180,E1 -1421.145,E2 -1421.145} C_VEL
LIN {X 0,Y 587.129,Z 679.77,A -85,B 0,C 180,E1 -1422.587,E2 -1422.587} C_VEL
LIN {X 0,Y 587.156,Z 677.816,A -85,B 0,C 180,E1 -1424.02,E2 -1424.02} C_VEL
LIN {X 0,Y 587.132,Z 674.567,A -85,B 0,C 180,E1 -1425.441,E2 -1425.441} C_VEL
LIN {X 0,Y 587.164,Z 670.04,A -85,B 0,C 180,E1 -1426.855,E2 -1426.855} C_VEL
LIN {X 0,Y 587.2,Z 664.118,A -85,B 0,C 180,E1 -1428.26,E2 -1428.26} C_VEL
LIN {X 0,Y 587.221,Z 656.674,A -85,B 0,C 180,E1 -1429.658,E2 -1429.658} C_VEL
LIN {X 0,Y 587.315,Z 648.768,A -85,B 0,C 180,E1 -1430.877,E2 -1430.877} C_VEL
LIN {X 0,Y 587.39,Z 639.317,A -85,B 0,C 180,E1 -1432.091,E2 -1432.091} C_VEL
LIN {X 0,Y 587.493,Z 628.295,A -85,B 0,C 180,E1 -1433.273,E2 -1433.273} C_VEL
LIN {X 0,Y 587.575,Z 616.425,A -85,B 0,C 180,E1 -1434.337,E2 -1434.337} C_VEL
LIN {X 0,Y 587.724,Z 603.686,A -85,B 0,C 180,E1 -1435.284,E2 -1435.284} C_VEL
LIN {X 0,Y 587.848,Z 591.168,A -85,B 0,C 180,E1 -1436.058,E2 -1436.058} C_VEL
LIN {X 0,Y 587.97,Z 577.591,A -85,B 0,C 180,E1 -1436.745,E2 -1436.745} C_VEL
LIN {X 0,Y 588.102,Z 562.51,A -85,B 0,C 180,E1 -1437.346,E2 -1437.346} C_VEL
LIN {X 0,Y 588.238,Z 547.209,A -85,B 0,C 180,E1 -1437.796,E2 -1437.796} C_VEL
LIN {X 0,Y 588.32,Z 532.129,A -85,B 0,C 180,E1 -1438.096,E2 -1438.096} C_VEL
LIN {X 0,Y 588.46,Z 373.714,A -85,B 0,C 180,E1 -1440.093,E2 -1440.093} C_VEL
LIN {X 0,Y 587.705,Z 369.909,A -85,B 0,C 180,E1 -1440.171,E2 -1440.171} C_VEL
LIN {X 0,Y 587.865,Z 349.632,A -85,B 0,C 180,E1 -1442.912,E2 -1442.912} C_VEL
LIN {X 0,Y 587.622,Z 343.438,A -85,B 0,C 180,E1 -1443.771,E2 -1443.771} C_VEL
LIN {X 0,Y 587.331,Z 341.951,A -85,B 0,C 180,E1 -1444.01,E2 -1444.01} C_VEL
LIN {X 0,Y 587.362,Z 341.947,A -85,B 0,C 180,E1 -1446.872,E2 -1446.872} C_VEL
LIN {X 0,Y 587.306,Z 341.948,A -85,B 0,C 180,E1 -1449.644,E2 -1449.644} C_VEL
LIN {X 0,Y 587.328,Z 341.945,A -85,B 0,C 180,E1 -1451.737,E2 -1451.737} C_VEL
LIN {X 0,Y 587.339,Z 341.952,A -85,B 0,C 180,E1 -1454.553,E2 -1454.553} C_VEL
LIN {X 0,Y 587.308,Z 341.947,A -85,B 0,C 180,E1 -1457.407,E2 -1457.407} C_VEL
LIN {X 0,Y 587.306,Z 341.948,A -85,B 0,C 180,E1 -1459.576,E2 -1459.576} C_VEL
LIN {X 0,Y 587.315,Z 341.948,A -85,B 0,C 180,E1 -1461.774,E2 -1461.774} C_VEL
LIN {X 0,Y 587.31,Z 341.95,A -85,B 0,C 180,E1 -1464.76,E2 -1464.76} C_VEL
LIN {X 0,Y 587.301,Z 341.95,A -85,B 0,C 180,E1 -1467.682,E2 -1467.682} C_VEL
LIN {X 0,Y 587.319,Z 341.951,A -85,B 0,C 180,E1 -1470.506,E2 -1470.506} C_VEL
LIN {X 0,Y 587.29,Z 341.949,A -85,B 0,C 180,E1 -1473.103,E2 -1473.103} C_VEL
LIN {X 0,Y 587.262,Z 341.954,A -85,B 0,C 180,E1 -1475.532,E2 -1475.532} C_VEL
LIN {X 0,Y 587.31,Z 341.951,A -85,B 0,C 180,E1 -1478.481,E2 -1478.481} C_VEL
LIN {X 0,Y 587.285,Z 341.95,A -85,B 0,C 180,E1 -1481.161,E2 -1481.161} C_VEL
LIN {X 0,Y 587.288,Z 341.958,A -85,B 0,C 180,E1 -1484.109,E2 -1484.109} C_VEL
LIN {X 0,Y 587.27,Z 341.951,A -85,B 0,C 180,E1 -1486.989,E2 -1486.989} C_VEL
LIN {X 0,Y 587.292,Z 341.959,A -85,B 0,C 180,E1 -1489.985,E2 -1489.985} C_VEL
LIN {X 0,Y 587.303,Z 341.951,A -85,B 0,C 180,E1 -1492.388,E2 -1492.388} C_VEL
LIN {X 0,Y 587.32,Z 341.952,A -85,B 0,C 180,E1 -1495.656,E2 -1495.656} C_VEL
LIN {X 0,Y 587.3,Z 341.953,A -85,B 0,C 180,E1 -1498.228,E2 -1498.228} C_VEL
LIN {X 0,Y 587.3,Z 341.949,A -85,B 0,C 180,E1 -1500.875,E2 -1500.875} C_VEL
LIN {X 0,Y 587.324,Z 341.954,A -85,B 0,C 180,E1 -1503.901,E2 -1503.901} C_VEL
LIN {X 0,Y 587.345,Z 342.177,A -85,B 0,C 180,E1 -1504.103,E2 -1504.103} C_VEL
LIN {X 0,Y 588.255,Z 346.855,A -85,B 0,C 180,E1 -1504.715,E2 -1504.715} C_VEL
LIN {X 0,Y 588.072,Z 370.263,A -85,B 0,C 180,E1 -1507.515,E2 -1507.515} C_VEL
LIN {X 0,Y 587.84,Z 396.356,A -85,B 0,C 180,E1 -1510.572,E2 -1510.572} C_VEL
LIN {X 0,Y 587.811,Z 399.136,A -85,B 0,C 180,E1 -1510.872,E2 -1510.872} C_VEL
LIN {X 0,Y 588.597,Z 403.498,A -85,B 0,C 180,E1 -1510.954,E2 -1510.954} C_VEL
LIN {X 0,Y 588.3,Z 565.363,A -85,B 0,C 180,E1 -1512.999,E2 -1512.999} C_VEL
LIN {X 0,Y 588.208,Z 580.677,A -85,B 0,C 180,E1 -1513.335,E2 -1513.335} C_VEL
LIN {X 0,Y 588.072,Z 596.022,A -85,B 0,C 180,E1 -1513.822,E2 -1513.822} C_VEL
LIN {X 0,Y 587.99,Z 609.745,A -85,B 0,C 180,E1 -1514.398,E2 -1514.398} C_VEL
LIN {X 0,Y 587.83,Z 623.223,A -85,B 0,C 180,E1 -1515.104,E2 -1515.104} C_VEL
LIN {X 0,Y 587.733,Z 636.101,A -85,B 0,C 180,E1 -1515.928,E2 -1515.928} C_VEL
LIN {X 0,Y 587.583,Z 648.276,A -85,B 0,C 180,E1 -1516.864,E2 -1516.864} C_VEL
LIN {X 0,Y 587.455,Z 659.739,A -85,B 0,C 180,E1 -1517.914,E2 -1517.914} C_VEL
LIN {X 0,Y 587.349,Z 669.382,A -85,B 0,C 180,E1 -1518.962,E2 -1518.962} C_VEL
LIN {X 0,Y 587.305,Z 678.849,A -85,B 0,C 180,E1 -1520.181,E2 -1520.181} C_VEL
LIN {X 0,Y 587.264,Z 686.726,A -85,B 0,C 180,E1 -1521.396,E2 -1521.396} C_VEL
LIN {X 0,Y 587.216,Z 694.084,A -85,B 0,C 180,E1 -1522.78,E2 -1522.78} C_VEL
LIN {X 0,Y 587.226,Z 699.92,A -85,B 0,C 180,E1 -1524.16,E2 -1524.16} C_VEL
LIN {X 0,Y 587.136,Z 703.381,A -85,B 0,C 180,E1 -1525.193,E2 -1525.193} C_VEL
LIN {X 0,Y 587.18,Z 706.886,A -85,B 0,C 180,E1 -1526.568,E2 -1526.568} C_VEL
LIN {X 0,Y 587.139,Z 709.192,A -85,B 0,C 180,E1 -1527.941,E2 -1527.941} C_VEL
LIN {X 0,Y 587.135,Z 710.349,A -85,B 0,C 180,E1 -1529.313,E2 -1529.313} C_VEL
LIN {X 0,Y 587.135,Z 710.35,A -85,B 0,C 180,E1 -1530.685,E2 -1530.685} C_VEL
LIN {X 0,Y 587.14,Z 709.194,A -85,B 0,C 180,E1 -1532.057,E2 -1532.057} C_VEL
LIN {X 0,Y 587.18,Z 706.888,A -85,B 0,C 180,E1 -1533.43,E2 -1533.43} C_VEL
LIN {X 0,Y 587.136,Z 703.387,A -85,B 0,C 180,E1 -1534.805,E2 -1534.805} C_VEL
LIN {X 0,Y 587.179,Z 698.613,A -85,B 0,C 180,E1 -1536.183,E2 -1536.183} C_VEL
LIN {X 0,Y 587.229,Z 692.43,A -85,B 0,C 180,E1 -1537.564,E2 -1537.564} C_VEL
LIN {X 0,Y 587.265,Z 684.658,A -85,B 0,C 180,E1 -1538.949,E2 -1538.949} C_VEL
LIN {X 0,Y 587.352,Z 676.378,A -85,B 0,C 180,E1 -1540.164,E2 -1540.164} C_VEL
LIN {X 0,Y 587.398,Z 666.405,A -85,B 0,C 180,E1 -1541.384,E2 -1541.384} C_VEL
LIN {X 0,Y 587.521,Z 656.203,A -85,B 0,C 180,E1 -1542.433,E2 -1542.433} C_VEL
LIN {X 0,Y 587.628,Z 644.033,A -85,B 0,C 180,E1 -1543.485,E2 -1543.485} C_VEL
LIN {X 0,Y 587.771,Z 631.075,A -85,B 0,C 180,E1 -1544.415,E2 -1544.415} C_VEL
LIN {X 0,Y 587.886,Z 616.89,A -85,B 0,C 180,E1 -1545.247,E2 -1545.247} C_VEL
LIN {X 0,Y 588.048,Z 602.827,A -85,B 0,C 180,E1 -1545.909,E2 -1545.909} C_VEL
LIN {X 0,Y 588.165,Z 588.342,A -85,B 0,C 180,E1 -1546.441,E2 -1546.441} C_VEL
LIN {X 0,Y 588.264,Z 572.506,A -85,B 0,C 180,E1 -1546.862,E2 -1546.862} C_VEL
LIN {X 0,Y 588.34,Z 556.486,A -85,B 0,C 180,E1 -1547.131,E2 -1547.131} C_VEL
LIN {X 0,Y 588.503,Z 402.481,A -85,B 0,C 180,E1 -1549.062,E2 -1549.062} C_VEL
LIN {X 0,Y 587.802,Z 398.78,A -85,B 0,C 180,E1 -1549.147,E2 -1549.147} C_VEL
LIN {X 0,Y 588.03,Z 373.403,A -85,B 0,C 180,E1 -1552.114,E2 -1552.114} C_VEL
LIN {X 0,Y 588.213,Z 351.188,A -85,B 0,C 180,E1 -1554.763,E2 -1554.763} C_VEL
LIN {X 0,Y 588.09,Z 345.312,A -85,B 0,C 180,E1 -1555.48,E2 -1555.48} C_VEL
LIN {X 0,Y 587.315,Z 341.954,A -85,B 0,C 180,E1 -1555.947,E2 -1555.947} C_VEL
LIN {X 0,Y 587.334,Z 341.945,A -85,B 0,C 180,E1 -1559.131,E2 -1559.131} C_VEL
LIN {X 0,Y 587.33,Z 341.948,A -85,B 0,C 180,E1 -1561.833,E2 -1561.833} C_VEL
LIN {X 0,Y 587.323,Z 341.953,A -85,B 0,C 180,E1 -1564.344,E2 -1564.344} C_VEL
LIN {X 0,Y 587.309,Z 341.948,A -85,B 0,C 180,E1 -1567.609,E2 -1567.609} C_VEL
LIN {X 0,Y 587.295,Z 341.958,A -85,B 0,C 180,E1 -1570.254,E2 -1570.254} C_VEL
LIN {X 0,Y 587.277,Z 341.95,A -85,B 0,C 180,E1 -1573.008,E2 -1573.008} C_VEL
LIN {X 0,Y 587.292,Z 341.954,A -85,B 0,C 180,E1 -1575.888,E2 -1575.888} C_VEL
LIN {X 0,Y 587.294,Z 341.948,A -85,B 0,C 180,E1 -1578.927,E2 -1578.927} C_VEL
LIN {X 0,Y 587.3,Z 341.949,A -85,B 0,C 180,E1 -1581.518,E2 -1581.518} C_VEL
LIN {X 0,Y 587.265,Z 341.962,A -85,B 0,C 180,E1 -1584.098,E2 -1584.098} C_VEL
LIN {X 0,Y 587.314,Z 341.949,A -85,B 0,C 180,E1 -1586.602,E2 -1586.602} C_VEL
LIN {X 0,Y 587.313,Z 341.947,A -85,B 0,C 180,E1 -1589.491,E2 -1589.491} C_VEL
LIN {X 0,Y 587.283,Z 341.956,A -85,B 0,C 180,E1 -1592.317,E2 -1592.317} C_VEL
LIN {X 0,Y 587.292,Z 341.948,A -85,B 0,C 180,E1 -1595.239,E2 -1595.239} C_VEL
LIN {X 0,Y 587.289,Z 341.957,A -85,B 0,C 180,E1 -1598.225,E2 -1598.225} C_VEL
LIN {X 0,Y 587.309,Z 341.946,A -85,B 0,C 180,E1 -1601.15,E2 -1601.15} C_VEL
LIN {X 0,Y 587.281,Z 341.96,A -85,B 0,C 180,E1 -1604.024,E2 -1604.024} C_VEL
LIN {X 0,Y 587.333,Z 341.952,A -85,B 0,C 180,E1 -1606.154,E2 -1606.154} C_VEL
LIN {X 0,Y 587.321,Z 341.945,A -85,B 0,C 180,E1 -1608.962,E2 -1608.962} C_VEL
LIN {X 0,Y 587.319,Z 341.95,A -85,B 0,C 180,E1 -1611.744,E2 -1611.744} C_VEL
LIN {X 0,Y 587.319,Z 341.948,A -85,B 0,C 180,E1 -1614.507,E2 -1614.507} C_VEL
LIN {X 0,Y 587.32,Z 341.945,A -85,B 0,C 180,E1 -1617.257,E2 -1617.257} C_VEL
LIN {X 0,Y 587.367,Z 341.95,A -85,B 0,C 180,E1 -1620,E2 -1620} C_VEL
LIN {X 0,Y 587.319,Z 341.945,A -85,B 0,C 180,E1 -1622.744,E2 -1622.744} C_VEL
LIN {X 0,Y 587.313,Z 341.948,A -85,B 0,C 180,E1 -1625.494,E2 -1625.494} C_VEL
LIN {X 0,Y 587.318,Z 341.951,A -85,B 0,C 180,E1 -1628.256,E2 -1628.256} C_VEL
LIN {X 0,Y 587.299,Z 341.948,A -85,B 0,C 180,E1 -1631.117,E2 -1631.117} C_VEL
LIN {X 0,Y 587.333,Z 341.952,A -85,B 0,C 180,E1 -1633.847,E2 -1633.847} C_VEL
LIN {X 0,Y 587.27,Z 341.951,A -85,B 0,C 180,E1 -1636.794,E2 -1636.794} C_VEL
LIN {X 0,Y 587.275,Z 341.955,A -85,B 0,C 180,E1 -1638.278,E2 -1638.278} C_VEL
LIN {X 0,Y 586.616,Z 342.035,A -85,B 0,C 180,E1 -1638.85,E2 -1638.85} C_VEL
LIN {X 0,Y 583.762,Z 342.396,A -85,B 0,C 180,E1 -1639.778,E2 -1639.778} C_VEL
LIN {X 0,Y 581.354,Z 342.691,A -85,B 0,C 180,E1 -1640.525,E2 -1640.525} C_VEL
LIN {X 0,Y 580.335,Z 342.815,A -85,B 0,C 180,E1 -1641.102,E2 -1641.102} C_VEL
LIN {X 0,Y 580.26,Z 342.826,A -85,B 0,C 180,E1 -1641.297,E2 -1641.297} C_VEL
LIN {X 0,Y 580.244,Z 342.831,A -85,B 0,C 180,E1 -1643.56,E2 -1643.56} C_VEL
LIN {X 0,Y 580.242,Z 342.83,A -85,B 0,C 180,E1 -1646.328,E2 -1646.328} C_VEL
LIN {X 0,Y 580.241,Z 342.828,A -85,B 0,C 180,E1 -1649.302,E2 -1649.302} C_VEL
LIN {X 0,Y 580.28,Z 342.827,A -85,B 0,C 180,E1 -1652.202,E2 -1652.202} C_VEL
LIN {X 0,Y 580.262,Z 342.824,A -85,B 0,C 180,E1 -1654.698,E2 -1654.698} C_VEL
LIN {X 0,Y 580.259,Z 342.826,A -85,B 0,C 180,E1 -1657.272,E2 -1657.272} C_VEL
LIN {X 0,Y 580.272,Z 342.826,A -85,B 0,C 180,E1 -1660.271,E2 -1660.271} C_VEL
LIN {X 0,Y 580.24,Z 342.827,A -85,B 0,C 180,E1 -1662.71,E2 -1662.71} C_VEL
LIN {X 0,Y 580.241,Z 342.833,A -85,B 0,C 180,E1 -1665.612,E2 -1665.612} C_VEL
LIN {X 0,Y 580.242,Z 342.83,A -85,B 0,C 180,E1 -1668.23,E2 -1668.23} C_VEL
LIN {X 0,Y 580.255,Z 342.825,A -85,B 0,C 180,E1 -1670.965,E2 -1670.965} C_VEL
LIN {X 0,Y 580.232,Z 342.835,A -85,B 0,C 180,E1 -1673.596,E2 -1673.596} C_VEL
LIN {X 0,Y 580.297,Z 342.824,A -85,B 0,C 180,E1 -1676.146,E2 -1676.146} C_VEL
LIN {X 0,Y 580.262,Z 342.824,A -85,B 0,C 180,E1 -1678.615,E2 -1678.615} C_VEL
LIN {X 0,Y 580.246,Z 342.827,A -85,B 0,C 180,E1 -1681.023,E2 -1681.023} C_VEL
LIN {X 0,Y 580.26,Z 342.833,A -85,B 0,C 180,E1 -1683.673,E2 -1683.673} C_VEL
LIN {X 0,Y 580.262,Z 342.825,A -85,B 0,C 180,E1 -1686.443,E2 -1686.443} C_VEL
LIN {X 0,Y 580.263,Z 342.829,A -85,B 0,C 180,E1 -1689.438,E2 -1689.438} C_VEL
LIN {X 0,Y 580.247,Z 342.835,A -85,B 0,C 180,E1 -1691.646,E2 -1691.646} C_VEL
LIN {X 0,Y 580.271,Z 342.823,A -85,B 0,C 180,E1 -1694.548,E2 -1694.548} C_VEL
LIN {X 0,Y 580.253,Z 342.825,A -85,B 0,C 180,E1 -1696.697,E2 -1696.697} C_VEL
LIN {X 0,Y 580.291,Z 342.828,A -85,B 0,C 180,E1 -1699.534,E2 -1699.534} C_VEL
LIN {X 0,Y 580.266,Z 342.825,A -85,B 0,C 180,E1 -1702.345,E2 -1702.345} C_VEL
LIN {X 0,Y 580.314,Z 342.82,A -85,B 0,C 180,E1 -1705.138,E2 -1705.138} C_VEL
LIN {X 0,Y 580.34,Z 342.82,A -85,B 0,C 180,E1 -1707.919,E2 -1707.919} C_VEL
LIN {X 0,Y 580.351,Z 342.817,A -85,B 0,C 180,E1 -1710.001,E2 -1710.001} C_VEL
LIN {X 0,Y 580.311,Z 342.818,A -85,B 0,C 180,E1 -1712.778,E2 -1712.778} C_VEL
LIN {X 0,Y 580.31,Z 342.827,A -85,B 0,C 180,E1 -1715.561,E2 -1715.561} C_VEL
LIN {X 0,Y 580.307,Z 342.819,A -85,B 0,C 180,E1 -1718.357,E2 -1718.357} C_VEL
LIN {X 0,Y 580.307,Z 342.822,A -85,B 0,C 180,E1 -1721.192,E2 -1721.192} C_VEL
LIN {X 0,Y 580.293,Z 342.821,A -85,B 0,C 180,E1 -1724.328,E2 -1724.328} C_VEL
LIN {X 0,Y 580.238,Z 342.828,A -85,B 0,C 180,E1 -1726.9,E2 -1726.9} C_VEL
LIN {X 0,Y 580.282,Z 342.828,A -85,B 0,C 180,E1 -1729.824,E2 -1729.824} C_VEL
LIN {X 0,Y 580.257,Z 342.827,A -85,B 0,C 180,E1 -1732.054,E2 -1732.054} C_VEL
LIN {X 0,Y 580.292,Z 342.823,A -85,B 0,C 180,E1 -1735.081,E2 -1735.081} C_VEL
LIN {X 0,Y 580.252,Z 342.826,A -85,B 0,C 180,E1 -1738.189,E2 -1738.189} C_VEL
LIN {X 0,Y 580.274,Z 342.823,A -85,B 0,C 180,E1 -1740.692,E2 -1740.692} C_VEL
LIN {X 0,Y 580.307,Z 342.825,A -85,B 0,C 180,E1 -1743.316,E2 -1743.316} C_VEL
LIN {X 0,Y 580.235,Z 342.834,A -85,B 0,C 180,E1 -1745.754,E2 -1745.754} C_VEL
LIN {X 0,Y 580.288,Z 342.823,A -85,B 0,C 180,E1 -1748.147,E2 -1748.147} C_VEL
LIN {X 0,Y 580.298,Z 342.822,A -85,B 0,C 180,E1 -1750.844,E2 -1750.844} C_VEL
LIN {X 0,Y 580.274,Z 342.831,A -85,B 0,C 180,E1 -1753.659,E2 -1753.659} C_VEL
LIN {X 0,Y 580.247,Z 342.829,A -85,B 0,C 180,E1 -1756.613,E2 -1756.613} C_VEL
LIN {X 0,Y 580.303,Z 342.946,A -85,B 0,C 180,E1 -1757.947,E2 -1757.947} C_VEL
LIN {X 0,Y 580.96,Z 347.393,A -85,B 0,C 180,E1 -1758.594,E2 -1758.594} C_VEL
LIN {X 0,Y 580.794,Z 366.579,A -85,B 0,C 180,E1 -1761.228,E2 -1761.228} C_VEL
LIN {X 0,Y 580.751,Z 369.93,A -85,B 0,C 180,E1 -1761.684,E2 -1761.684} C_VEL
LIN {X 0,Y 581.855,Z 375.488,A -85,B 0,C 180,E1 -1761.795,E2 -1761.795} C_VEL
LIN {X 0,Y 581.525,Z 534.754,A -85,B 0,C 180,E1 -1763.83,E2 -1763.83} C_VEL
LIN {X 0,Y 581.405,Z 550.846,A -85,B 0,C 180,E1 -1764.184,E2 -1764.184} C_VEL
LIN {X 0,Y 581.25,Z 565.138,A -85,B 0,C 180,E1 -1764.64,E2 -1764.64} C_VEL
LIN {X 0,Y 581.123,Z 578.329,A -85,B 0,C 180,E1 -1765.19,E2 -1765.19} C_VEL
LIN {X 0,Y 580.91,Z 591.474,A -85,B 0,C 180,E1 -1765.871,E2 -1765.871} C_VEL
LIN {X 0,Y 580.807,Z 603.353,A -85,B 0,C 180,E1 -1766.609,E2 -1766.609} C_VEL
LIN {X 0,Y 580.636,Z 615.487,A -85,B 0,C 180,E1 -1767.512,E2 -1767.512} C_VEL
LIN {X 0,Y 580.485,Z 626.853,A -85,B 0,C 180,E1 -1768.525,E2 -1768.525} C_VEL
LIN {X 0,Y 580.392,Z 637.364,A -85,B 0,C 180,E1 -1769.632,E2 -1769.632} C_VEL
LIN {X 0,Y 580.282,Z 647.099,A -85,B 0,C 180,E1 -1770.858,E2 -1770.858} C_VEL
LIN {X 0,Y 580.206,Z 655.701,A -85,B 0,C 180,E1 -1772.16,E2 -1772.16} C_VEL
LIN {X 0,Y 580.136,Z 662.322,A -85,B 0,C 180,E1 -1773.369,E2 -1773.369} C_VEL
LIN {X 0,Y 580.096,Z 667.568,A -85,B 0,C 180,E1 -1774.526,E2 -1774.526} C_VEL
LIN {X 0,Y 580.086,Z 673.007,A -85,B 0,C 180,E1 -1776.054,E2 -1776.054} C_VEL
LIN {X 0,Y 580.063,Z 676.075,A -85,B 0,C 180,E1 -1777.188,E2 -1777.188} C_VEL
LIN {X 0,Y 580.053,Z 678.835,A -85,B 0,C 180,E1 -1778.685,E2 -1778.685} C_VEL
LIN {X 0,Y 580.021,Z 680.265,A -85,B 0,C 180,E1 -1780.167,E2 -1780.167} C_VEL
LIN {X 0,Y 580.036,Z 680.368,A -85,B 0,C 180,E1 -1781.637,E2 -1781.637} C_VEL
LIN {X 0,Y 580.043,Z 679.151,A -85,B 0,C 180,E1 -1783.176,E2 -1783.176} C_VEL
LIN {X 0,Y 580.038,Z 676.844,A -85,B 0,C 180,E1 -1784.54,E2 -1784.54} C_VEL
LIN {X 0,Y 580.087,Z 673.185,A -85,B 0,C 180,E1 -1785.977,E2 -1785.977} C_VEL
LIN {X 0,Y 580.108,Z 668.216,A -85,B 0,C 180,E1 -1787.404,E2 -1787.404} C_VEL
LIN {X 0,Y 580.167,Z 661.519,A -85,B 0,C 180,E1 -1788.878,E2 -1788.878} C_VEL
LIN {X 0,Y 580.216,Z 653.822,A -85,B 0,C 180,E1 -1790.236,E2 -1790.236} C_VEL
LIN {X 0,Y 580.277,Z 645.376,A -85,B 0,C 180,E1 -1791.468,E2 -1791.468} C_VEL
LIN {X 0,Y 580.417,Z 635.228,A -85,B 0,C 180,E1 -1792.695,E2 -1792.695} C_VEL
LIN {X 0,Y 580.519,Z 624.999,A -85,B 0,C 180,E1 -1793.745,E2 -1793.745} C_VEL
LIN {X 0,Y 580.684,Z 612.727,A -85,B 0,C 180,E1 -1794.792,E2 -1794.792} C_VEL
LIN {X 0,Y 580.869,Z 600.629,A -85,B 0,C 180,E1 -1795.663,E2 -1795.663} C_VEL
LIN {X 0,Y 581.001,Z 587.492,A -85,B 0,C 180,E1 -1796.446,E2 -1796.446} C_VEL
LIN {X 0,Y 581.164,Z 572.977,A -85,B 0,C 180,E1 -1797.14,E2 -1797.14} C_VEL
LIN {X 0,Y 581.304,Z 558.257,A -85,B 0,C 180,E1 -1797.683,E2 -1797.683} C_VEL
LIN {X 0,Y 581.45,Z 544.138,A -85,B 0,C 180,E1 -1798.073,E2 -1798.073} C_VEL
LIN {X 0,Y 581.529,Z 528.501,A -85,B 0,C 180,E1 -1798.355,E2 -1798.355} C_VEL
LIN {X 0,Y 581.797,Z 375.074,A -85,B 0,C 180,E1 -1800.303,E2 -1800.303} C_VEL
LIN {X 0,Y 580.775,Z 369.886,A -85,B 0,C 180,E1 -1800.411,E2 -1800.411} C_VEL
LIN {X 0,Y 580.956,Z 348.853,A -85,B 0,C 180,E1 -1803.294,E2 -1803.294} C_VEL
LIN {X 0,Y 580.753,Z 345.156,A -85,B 0,C 180,E1 -1803.816,E2 -1803.816} C_VEL
LIN {X 0,Y 580.273,Z 342.831,A -85,B 0,C 180,E1 -1804.167,E2 -1804.167} C_VEL
LIN {X 0,Y 580.33,Z 342.822,A -85,B 0,C 180,E1 -1806.956,E2 -1806.956} C_VEL
LIN {X 0,Y 580.26,Z 342.827,A -85,B 0,C 180,E1 -1809.762,E2 -1809.762} C_VEL
LIN {X 0,Y 580.3,Z 342.822,A -85,B 0,C 180,E1 -1811.881,E2 -1811.881} C_VEL
LIN {X 0,Y 580.286,Z 342.828,A -85,B 0,C 180,E1 -1814.734,E2 -1814.734} C_VEL
LIN {X 0,Y 580.266,Z 342.825,A -85,B 0,C 180,E1 -1817.625,E2 -1817.625} C_VEL
LIN {X 0,Y 580.282,Z 342.824,A -85,B 0,C 180,E1 -1819.823,E2 -1819.823} C_VEL
LIN {X 0,Y 580.267,Z 342.829,A -85,B 0,C 180,E1 -1822.053,E2 -1822.053} C_VEL
LIN {X 0,Y 580.278,Z 342.823,A -85,B 0,C 180,E1 -1825.081,E2 -1825.081} C_VEL
LIN {X 0,Y 580.25,Z 342.83,A -85,B 0,C 180,E1 -1827.849,E2 -1827.849} C_VEL
LIN {X 0,Y 580.269,Z 342.827,A -85,B 0,C 180,E1 -1830.691,E2 -1830.691} C_VEL
LIN {X 0,Y 580.273,Z 342.823,A -85,B 0,C 180,E1 -1833.311,E2 -1833.311} C_VEL
LIN {X 0,Y 580.221,Z 342.834,A -85,B 0,C 180,E1 -1835.752,E2 -1835.752} C_VEL
LIN {X 0,Y 580.277,Z 342.833,A -85,B 0,C 180,E1 -1838.147,E2 -1838.147} C_VEL
LIN {X 0,Y 580.236,Z 342.828,A -85,B 0,C 180,E1 -1840.849,E2 -1840.849} C_VEL
LIN {X 0,Y 580.225,Z 342.833,A -85,B 0,C 180,E1 -1843.663,E2 -1843.663} C_VEL
LIN {X 0,Y 580.22,Z 342.831,A -85,B 0,C 180,E1 -1846.615,E2 -1846.615} C_VEL
LIN {X 0,Y 580.234,Z 342.828,A -85,B 0,C 180,E1 -1849.15,E2 -1849.15} C_VEL
LIN {X 0,Y 580.269,Z 342.834,A -85,B 0,C 180,E1 -1851.93,E2 -1851.93} C_VEL
LIN {X 0,Y 580.216,Z 342.833,A -85,B 0,C 180,E1 -1854.449,E2 -1854.449} C_VEL
LIN {X 0,Y 580.242,Z 342.829,A -85,B 0,C 180,E1 -1856.971,E2 -1856.971} C_VEL
LIN {X 0,Y 580.274,Z 342.829,A -85,B 0,C 180,E1 -1859.423,E2 -1859.423} C_VEL
LIN {X 0,Y 580.242,Z 342.834,A -85,B 0,C 180,E1 -1862.152,E2 -1862.152} C_VEL
LIN {X 0,Y 580.299,Z 342.912,A -85,B 0,C 180,E1 -1863.856,E2 -1863.856} C_VEL
LIN {X 0,Y 581.447,Z 348.414,A -85,B 0,C 180,E1 -1864.589,E2 -1864.589} C_VEL
LIN {X 0,Y 581.209,Z 371.824,A -85,B 0,C 180,E1 -1867.422,E2 -1867.422} C_VEL
LIN {X 0,Y 580.924,Z 396.542,A -85,B 0,C 180,E1 -1870.353,E2 -1870.353} C_VEL
LIN {X 0,Y 580.899,Z 398.898,A -85,B 0,C 180,E1 -1870.63,E2 -1870.63} C_VEL
LIN {X 0,Y 581.88,Z 404.68,A -85,B 0,C 180,E1 -1870.74,E2 -1870.74} C_VEL
LIN {X 0,Y 581.531,Z 565.452,A -85,B 0,C 180,E1 -1872.797,E2 -1872.797} C_VEL
LIN {X 0,Y 581.414,Z 580.676,A -85,B 0,C 180,E1 -1873.135,E2 -1873.135} C_VEL
LIN {X 0,Y 581.234,Z 596.02,A -85,B 0,C 180,E1 -1873.626,E2 -1873.626} C_VEL
LIN {X 0,Y 581.125,Z 609.748,A -85,B 0,C 180,E1 -1874.209,E2 -1874.209} C_VEL
LIN {X 0,Y 580.945,Z 623.225,A -85,B 0,C 180,E1 -1874.923,E2 -1874.923} C_VEL
LIN {X 0,Y 580.797,Z 636.466,A -85,B 0,C 180,E1 -1875.782,E2 -1875.782} C_VEL
LIN {X 0,Y 580.609,Z 648.277,A -85,B 0,C 180,E1 -1876.703,E2 -1876.703} C_VEL
LIN {X 0,Y 580.48,Z 659.74,A -85,B 0,C 180,E1 -1877.767,E2 -1877.767} C_VEL
LIN {X 0,Y 580.308,Z 670.452,A -85,B 0,C 180,E1 -1878.953,E2 -1878.953} C_VEL
LIN {X 0,Y 580.269,Z 678.85,A -85,B 0,C 180,E1 -1880.061,E2 -1880.061} C_VEL
LIN {X 0,Y 580.214,Z 686.727,A -85,B 0,C 180,E1 -1881.29,E2 -1881.29} C_VEL
LIN {X 0,Y 580.131,Z 694.084,A -85,B 0,C 180,E1 -1882.691,E2 -1882.691} C_VEL
LIN {X 0,Y 580.131,Z 699.92,A -85,B 0,C 180,E1 -1884.089,E2 -1884.089} C_VEL
LIN {X 0,Y 580.041,Z 703.382,A -85,B 0,C 180,E1 -1885.134,E2 -1885.134} C_VEL
LIN {X 0,Y 580.105,Z 706.886,A -85,B 0,C 180,E1 -1886.526,E2 -1886.526} C_VEL
LIN {X 0,Y 580.038,Z 709.192,A -85,B 0,C 180,E1 -1887.916,E2 -1887.916} C_VEL
LIN {X 0,Y 580.036,Z 710.349,A -85,B 0,C 180,E1 -1889.305,E2 -1889.305} C_VEL
LIN {X 0,Y 580.036,Z 710.349,A -85,B 0,C 180,E1 -1890.693,E2 -1890.693} C_VEL
LIN {X 0,Y 580.038,Z 709.193,A -85,B 0,C 180,E1 -1892.082,E2 -1892.082} C_VEL
LIN {X 0,Y 580.105,Z 706.889,A -85,B 0,C 180,E1 -1893.472,E2 -1893.472} C_VEL
LIN {X 0,Y 580.041,Z 703.388,A -85,B 0,C 180,E1 -1894.864,E2 -1894.864} C_VEL
LIN {X 0,Y 580.092,Z 698.613,A -85,B 0,C 180,E1 -1896.259,E2 -1896.259} C_VEL
LIN {X 0,Y 580.164,Z 692.429,A -85,B 0,C 180,E1 -1897.656,E2 -1897.656} C_VEL
LIN {X 0,Y 580.206,Z 684.657,A -85,B 0,C 180,E1 -1899.059,E2 -1899.059} C_VEL
LIN {X 0,Y 580.309,Z 676.378,A -85,B 0,C 180,E1 -1900.289,E2 -1900.289} C_VEL
LIN {X 0,Y 580.381,Z 666.405,A -85,B 0,C 180,E1 -1901.524,E2 -1901.524} C_VEL
LIN {X 0,Y 580.54,Z 656.202,A -85,B 0,C 180,E1 -1902.585,E2 -1902.585} C_VEL
LIN {X 0,Y 580.677,Z 644.034,A -85,B 0,C 180,E1 -1903.65,E2 -1903.65} C_VEL
LIN {X 0,Y 580.871,Z 630.545,A -85,B 0,C 180,E1 -1904.624,E2 -1904.624} C_VEL
LIN {X 0,Y 581.016,Z 616.892,A -85,B 0,C 180,E1 -1905.432,E2 -1905.432} C_VEL
LIN {X 0,Y 581.198,Z 602.828,A -85,B 0,C 180,E1 -1906.102,E2 -1906.102} C_VEL
LIN {X 0,Y 581.354,Z 588.342,A -85,B 0,C 180,E1 -1906.639,E2 -1906.639} C_VEL
LIN {X 0,Y 581.483,Z 573.109,A -85,B 0,C 180,E1 -1907.051,E2 -1907.051} C_VEL
LIN {X 0,Y 581.548,Z 557.615,A -85,B 0,C 180,E1 -1907.322,E2 -1907.322} C_VEL
LIN {X 0,Y 581.811,Z 403.714,A -85,B 0,C 180,E1 -1909.275,E2 -1909.275} C_VEL
LIN {X 0,Y 580.918,Z 398.769,A -85,B 0,C 180,E1 -1909.385,E2 -1909.385} C_VEL
LIN {X 0,Y 581.176,Z 374.964,A -85,B 0,C 180,E1 -1912.202,E2 -1912.202} C_VEL
LIN {X 0,Y 581.411,Z 351.554,A -85,B 0,C 180,E1 -1915.027,E2 -1915.027} C_VEL
LIN {X 0,Y 581.212,Z 346.872,A -85,B 0,C 180,E1 -1915.611,E2 -1915.611} C_VEL
LIN {X 0,Y 580.271,Z 342.832,A -85,B 0,C 180,E1 -1916.171,E2 -1916.171} C_VEL
LIN {X 0,Y 580.271,Z 342.825,A -85,B 0,C 180,E1 -1919.304,E2 -1919.304} C_VEL
LIN {X 0,Y 580.286,Z 342.831,A -85,B 0,C 180,E1 -1922.2,E2 -1922.2} C_VEL
LIN {X 0,Y 580.265,Z 342.827,A -85,B 0,C 180,E1 -1924.696,E2 -1924.696} C_VEL
LIN {X 0,Y 580.262,Z 342.824,A -85,B 0,C 180,E1 -1927.269,E2 -1927.269} C_VEL
LIN {X 0,Y 580.274,Z 342.832,A -85,B 0,C 180,E1 -1930.269,E2 -1930.269} C_VEL
LIN {X 0,Y 580.251,Z 342.828,A -85,B 0,C 180,E1 -1932.707,E2 -1932.707} C_VEL
LIN {X 0,Y 580.239,Z 342.829,A -85,B 0,C 180,E1 -1935.61,E2 -1935.61} C_VEL
LIN {X 0,Y 580.236,Z 342.837,A -85,B 0,C 180,E1 -1938.227,E2 -1938.227} C_VEL
LIN {X 0,Y 580.252,Z 342.826,A -85,B 0,C 180,E1 -1940.963,E2 -1940.963} C_VEL
LIN {X 0,Y 580.225,Z 342.831,A -85,B 0,C 180,E1 -1943.593,E2 -1943.593} C_VEL
LIN {X 0,Y 580.293,Z 342.831,A -85,B 0,C 180,E1 -1946.144,E2 -1946.144} C_VEL
LIN {X 0,Y 580.252,Z 342.828,A -85,B 0,C 180,E1 -1948.613,E2 -1948.613} C_VEL
LIN {X 0,Y 580.235,Z 342.827,A -85,B 0,C 180,E1 -1951.021,E2 -1951.021} C_VEL
LIN {X 0,Y 580.242,Z 342.83,A -85,B 0,C 180,E1 -1953.672,E2 -1953.672} C_VEL
LIN {X 0,Y 580.246,Z 342.831,A -85,B 0,C 180,E1 -1956.441,E2 -1956.441} C_VEL
LIN {X 0,Y 580.239,Z 342.828,A -85,B 0,C 180,E1 -1959.436,E2 -1959.436} C_VEL
LIN {X 0,Y 580.231,Z 342.831,A -85,B 0,C 180,E1 -1961.644,E2 -1961.644} C_VEL
LIN {X 0,Y 580.253,Z 342.828,A -85,B 0,C 180,E1 -1964.546,E2 -1964.546} C_VEL
LIN {X 0,Y 580.224,Z 342.83,A -85,B 0,C 180,E1 -1966.695,E2 -1966.695} C_VEL
LIN {X 0,Y 580.289,Z 342.821,A -85,B 0,C 180,E1 -1968.827,E2 -1968.827} C_VEL
LIN {X 0,Y 580.286,Z 342.825,A -85,B 0,C 180,E1 -1971.643,E2 -1971.643} C_VEL
LIN {X 0,Y 580.29,Z 342.824,A -85,B 0,C 180,E1 -1974.44,E2 -1974.44} C_VEL
LIN {X 0,Y 580.329,Z 342.824,A -85,B 0,C 180,E1 -1977.918,E2 -1977.918} C_VEL
LIN {X 0,Y 580.335,Z 342.826,A -85,B 0,C 180,E1 -1980,E2 -1980} C_VEL
LIN {X 0,Y 580.287,Z 342.821,A -85,B 0,C 180,E1 -1982.777,E2 -1982.777} C_VEL
LIN {X 0,Y 580.282,Z 342.825,A -85,B 0,C 180,E1 -1985.56,E2 -1985.56} C_VEL
LIN {X 0,Y 580.285,Z 342.825,A -85,B 0,C 180,E1 -1988.357,E2 -1988.357} C_VEL
LIN {X 0,Y 580.251,Z 342.826,A -85,B 0,C 180,E1 -1991.174,E2 -1991.174} C_VEL
LIN {X 0,Y 580.294,Z 342.829,A -85,B 0,C 180,E1 -1994.018,E2 -1994.018} C_VEL
LIN {X 0,Y 580.234,Z 342.827,A -85,B 0,C 180,E1 -1996.9,E2 -1996.9} C_VEL
LIN {X 0,Y 580.259,Z 342.833,A -85,B 0,C 180,E1 -1999.824,E2 -1999.824} C_VEL
LIN {X 0,Y 580.26,Z 342.826,A -85,B 0,C 180,E1 -2001.297,E2 -2001.297} C_VEL
LIN {X 0,Y 579.607,Z 342.915,A -85,B 0,C 180,E1 -2001.876,E2 -2001.876} C_VEL
LIN {X 0,Y 576.73,Z 343.273,A -85,B 0,C 180,E1 -2002.816,E2 -2002.816} C_VEL
LIN {X 0,Y 574.297,Z 343.575,A -85,B 0,C 180,E1 -2003.572,E2 -2003.572} C_VEL
LIN {X 0,Y 573.265,Z 343.702,A -85,B 0,C 180,E1 -2004.156,E2 -2004.156} C_VEL
LIN {X 0,Y 573.189,Z 343.708,A -85,B 0,C 180,E1 -2004.354,E2 -2004.354} C_VEL
LIN {X 0,Y 573.17,Z 343.707,A -85,B 0,C 180,E1 -2006.98,E2 -2006.98} C_VEL
LIN {X 0,Y 573.194,Z 343.708,A -85,B 0,C 180,E1 -2009.482,E2 -2009.482} C_VEL
LIN {X 0,Y 573.233,Z 343.704,A -85,B 0,C 180,E1 -2012.228,E2 -2012.228} C_VEL
LIN {X 0,Y 573.208,Z 343.703,A -85,B 0,C 180,E1 -2014.77,E2 -2014.77} C_VEL
LIN {X 0,Y 573.209,Z 343.712,A -85,B 0,C 180,E1 -2017.81,E2 -2017.81} C_VEL
LIN {X 0,Y 573.235,Z 343.7,A -85,B 0,C 180,E1 -2020.526,E2 -2020.526} C_VEL
LIN {X 0,Y 573.194,Z 343.712,A -85,B 0,C 180,E1 -2023.666,E2 -2023.666} C_VEL
LIN {X 0,Y 573.19,Z 343.705,A -85,B 0,C 180,E1 -2026.638,E2 -2026.638} C_VEL
LIN {X 0,Y 573.238,Z 343.704,A -85,B 0,C 180,E1 -2029.476,E2 -2029.476} C_VEL
LIN {X 0,Y 573.213,Z 343.706,A -85,B 0,C 180,E1 -2032.193,E2 -2032.193} C_VEL
LIN {X 0,Y 573.213,Z 343.704,A -85,B 0,C 180,E1 -2035.233,E2 -2035.233} C_VEL
LIN {X 0,Y 573.242,Z 343.709,A -85,B 0,C 180,E1 -2037.774,E2 -2037.774} C_VEL
LIN {X 0,Y 573.221,Z 343.701,A -85,B 0,C 180,E1 -2040.633,E2 -2040.633} C_VEL
LIN {X 0,Y 573.201,Z 343.71,A -85,B 0,C 180,E1 -2043.516,E2 -2043.516} C_VEL
LIN {X 0,Y 573.214,Z 343.706,A -85,B 0,C 180,E1 -2046.135,E2 -2046.135} C_VEL
LIN {X 0,Y 573.245,Z 343.7,A -85,B 0,C 180,E1 -2049.175,E2 -2049.175} C_VEL
LIN {X 0,Y 573.203,Z 343.708,A -85,B 0,C 180,E1 -2051.412,E2 -2051.412} C_VEL
LIN {X 0,Y 573.21,Z 343.704,A -85,B 0,C 180,E1 -2054.353,E2 -2054.353} C_VEL
LIN {X 0,Y 573.214,Z 343.702,A -85,B 0,C 180,E1 -2056.53,E2 -2056.53} C_VEL
LIN {X 0,Y 573.26,Z 343.702,A -85,B 0,C 180,E1 -2059.404,E2 -2059.404} C_VEL
LIN {X 0,Y 573.222,Z 343.703,A -85,B 0,C 180,E1 -2062.25,E2 -2062.25} C_VEL
LIN {X 0,Y 573.287,Z 343.695,A -85,B 0,C 180,E1 -2065.078,E2 -2065.078} C_VEL
LIN {X 0,Y 573.311,Z 343.696,A -85,B 0,C 180,E1 -2067.893,E2 -2067.893} C_VEL
LIN {X 0,Y 573.32,Z 343.693,A -85,B 0,C 180,E1 -2070.001,E2 -2070.001} C_VEL
LIN {X 0,Y 573.279,Z 343.694,A -85,B 0,C 180,E1 -2072.812,E2 -2072.812} C_VEL
LIN {X 0,Y 573.278,Z 343.705,A -85,B 0,C 180,E1 -2075.629,E2 -2075.629} C_VEL
LIN {X 0,Y 573.25,Z 343.698,A -85,B 0,C 180,E1 -2078.461,E2 -2078.461} C_VEL
LIN {X 0,Y 573.278,Z 343.699,A -85,B 0,C 180,E1 -2081.313,E2 -2081.313} C_VEL
LIN {X 0,Y 573.269,Z 343.695,A -85,B 0,C 180,E1 -2084.418,E2 -2084.418} C_VEL
LIN {X 0,Y 573.187,Z 343.708,A -85,B 0,C 180,E1 -2087.115,E2 -2087.115} C_VEL
LIN {X 0,Y 573.272,Z 343.701,A -85,B 0,C 180,E1 -2089.331,E2 -2089.331} C_VEL
LIN {X 0,Y 573.224,Z 343.701,A -85,B 0,C 180,E1 -2092.339,E2 -2092.339} C_VEL
LIN {X 0,Y 573.238,Z 343.707,A -85,B 0,C 180,E1 -2095.412,E2 -2095.412} C_VEL
LIN {X 0,Y 573.211,Z 343.702,A -85,B 0,C 180,E1 -2098.567,E2 -2098.567} C_VEL
LIN {X 0,Y 573.223,Z 343.703,A -85,B 0,C 180,E1 -2100.994,E2 -2100.994} C_VEL
LIN {X 0,Y 573.27,Z 343.706,A -85,B 0,C 180,E1 -2103.524,E2 -2103.524} C_VEL
LIN {X 0,Y 573.194,Z 343.708,A -85,B 0,C 180,E1 -2106.054,E2 -2106.054} C_VEL
LIN {X 0,Y 573.239,Z 343.7,A -85,B 0,C 180,E1 -2108.703,E2 -2108.703} C_VEL
LIN {X 0,Y 573.228,Z 343.71,A -85,B 0,C 180,E1 -2111.592,E2 -2111.592} C_VEL
LIN {X 0,Y 573.228,Z 343.702,A -85,B 0,C 180,E1 -2114.335,E2 -2114.335} C_VEL
LIN {X 0,Y 573.241,Z 343.709,A -85,B 0,C 180,E1 -2117.359,E2 -2117.359} C_VEL
LIN {X 0,Y 573.263,Z 343.712,A -85,B 0,C 180,E1 -2117.755,E2 -2117.755} C_VEL
LIN {X 0,Y 574.064,Z 349.576,A -85,B 0,C 180,E1 -2118.616,E2 -2118.616} C_VEL
LIN {X 0,Y 573.855,Z 367.617,A -85,B 0,C 180,E1 -2121.122,E2 -2121.122} C_VEL
LIN {X 0,Y 573.852,Z 370.09,A -85,B 0,C 180,E1 -2121.445,E2 -2121.445} C_VEL
LIN {X 0,Y 575.154,Z 377.045,A -85,B 0,C 180,E1 -2121.582,E2 -2121.582} C_VEL
LIN {X 0,Y 574.753,Z 534.221,A -85,B 0,C 180,E1 -2123.611,E2 -2123.611} C_VEL
LIN {X 0,Y 574.598,Z 550.585,A -85,B 0,C 180,E1 -2123.971,E2 -2123.971} C_VEL
LIN {X 0,Y 574.422,Z 565.882,A -85,B 0,C 180,E1 -2124.468,E2 -2124.468} C_VEL
LIN {X 0,Y 574.249,Z 579.066,A -85,B 0,C 180,E1 -2125.032,E2 -2125.032} C_VEL
LIN {X 0,Y 574.082,Z 590.474,A -85,B 0,C 180,E1 -2125.628,E2 -2125.628} C_VEL
LIN {X 0,Y 573.892,Z 602.658,A -85,B 0,C 180,E1 -2126.382,E2 -2126.382} C_VEL
LIN {X 0,Y 573.664,Z 615.92,A -85,B 0,C 180,E1 -2127.381,E2 -2127.381} C_VEL
LIN {X 0,Y 573.48,Z 628.242,A -85,B 0,C 180,E1 -2128.508,E2 -2128.508} C_VEL
LIN {X 0,Y 573.345,Z 638.501,A -85,B 0,C 180,E1 -2129.626,E2 -2129.626} C_VEL
LIN {X 0,Y 573.234,Z 647.832,A -85,B 0,C 180,E1 -2130.833,E2 -2130.833} C_VEL
LIN {X 0,Y 573.129,Z 656.711,A -85,B 0,C 180,E1 -2132.226,E2 -2132.226} C_VEL
LIN {X 0,Y 573.077,Z 663.619,A -85,B 0,C 180,E1 -2133.541,E2 -2133.541} C_VEL
LIN {X 0,Y 573.02,Z 669.381,A -85,B 0,C 180,E1 -2134.912,E2 -2134.912} C_VEL
LIN {X 0,Y 573.008,Z 673.404,A -85,B 0,C 180,E1 -2136.124,E2 -2136.124} C_VEL
LIN {X 0,Y 572.943,Z 677.134,A -85,B 0,C 180,E1 -2137.65,E2 -2137.65} C_VEL
LIN {X 0,Y 572.942,Z 679.456,A -85,B 0,C 180,E1 -2139.162,E2 -2139.162} C_VEL
LIN {X 0,Y 572.971,Z 680.456,A -85,B 0,C 180,E1 -2140.818,E2 -2140.818} C_VEL
LIN {X 0,Y 572.943,Z 680.129,A -85,B 0,C 180,E1 -2142.142,E2 -2142.142} C_VEL
LIN {X 0,Y 572.938,Z 678.582,A -85,B 0,C 180,E1 -2143.612,E2 -2143.612} C_VEL
LIN {X 0,Y 572.945,Z 675.768,A -85,B 0,C 180,E1 -2145.072,E2 -2145.072} C_VEL
LIN {X 0,Y 573.012,Z 671.688,A -85,B 0,C 180,E1 -2146.524,E2 -2146.524} C_VEL
LIN {X 0,Y 573.04,Z 666.232,A -85,B 0,C 180,E1 -2147.966,E2 -2147.966} C_VEL
LIN {X 0,Y 573.078,Z 659.35,A -85,B 0,C 180,E1 -2149.4,E2 -2149.4} C_VEL
LIN {X 0,Y 573.17,Z 651.922,A -85,B 0,C 180,E1 -2150.65,E2 -2150.65} C_VEL
LIN {X 0,Y 573.328,Z 643.098,A -85,B 0,C 180,E1 -2151.896,E2 -2151.896} C_VEL
LIN {X 0,Y 573.413,Z 632.784,A -85,B 0,C 180,E1 -2153.11,E2 -2153.11} C_VEL
LIN {X 0,Y 573.604,Z 621.777,A -85,B 0,C 180,E1 -2154.198,E2 -2154.198} C_VEL
LIN {X 0,Y 573.766,Z 610.062,A -85,B 0,C 180,E1 -2155.169,E2 -2155.169} C_VEL
LIN {X 0,Y 573.963,Z 597.431,A -85,B 0,C 180,E1 -2156.05,E2 -2156.05} C_VEL
LIN {X 0,Y 574.201,Z 583.505,A -85,B 0,C 180,E1 -2156.842,E2 -2156.842} C_VEL
LIN {X 0,Y 574.382,Z 568.99,A -85,B 0,C 180,E1 -2157.501,E2 -2157.501} C_VEL
LIN {X 0,Y 574.554,Z 553.692,A -85,B 0,C 180,E1 -2158.028,E2 -2158.028} C_VEL
LIN {X 0,Y 574.732,Z 538.397,A -85,B 0,C 180,E1 -2158.401,E2 -2158.401} C_VEL
LIN {X 0,Y 574.809,Z 517.422,A -85,B 0,C 180,E1 -2158.708,E2 -2158.708} C_VEL
LIN {X 0,Y 575.105,Z 375.904,A -85,B 0,C 180,E1 -2160.525,E2 -2160.525} C_VEL
LIN {X 0,Y 573.841,Z 369.867,A -85,B 0,C 180,E1 -2160.658,E2 -2160.658} C_VEL
LIN {X 0,Y 574.068,Z 349.325,A -85,B 0,C 180,E1 -2163.509,E2 -2163.509} C_VEL
LIN {X 0,Y 573.391,Z 344.506,A -85,B 0,C 180,E1 -2164.217,E2 -2164.217} C_VEL
LIN {X 0,Y 573.25,Z 343.706,A -85,B 0,C 180,E1 -2164.35,E2 -2164.35} C_VEL
LIN {X 0,Y 573.295,Z 343.698,A -85,B 0,C 180,E1 -2167.041,E2 -2167.041} C_VEL
LIN {X 0,Y 573.215,Z 343.705,A -85,B 0,C 180,E1 -2169.884,E2 -2169.884} C_VEL
LIN {X 0,Y 573.27,Z 343.699,A -85,B 0,C 180,E1 -2172.029,E2 -2172.029} C_VEL
LIN {X 0,Y 573.233,Z 343.704,A -85,B 0,C 180,E1 -2174.92,E2 -2174.92} C_VEL
LIN {X 0,Y 573.225,Z 343.704,A -85,B 0,C 180,E1 -2177.849,E2 -2177.849} C_VEL
LIN {X 0,Y 573.239,Z 343.705,A -85,B 0,C 180,E1 -2180.077,E2 -2180.077} C_VEL
LIN {X 0,Y 573.232,Z 343.71,A -85,B 0,C 180,E1 -2182.338,E2 -2182.338} C_VEL
LIN {X 0,Y 573.225,Z 343.701,A -85,B 0,C 180,E1 -2185.411,E2 -2185.411} C_VEL
LIN {X 0,Y 573.187,Z 343.711,A -85,B 0,C 180,E1 -2188.567,E2 -2188.567} C_VEL
LIN {X 0,Y 573.218,Z 343.703,A -85,B 0,C 180,E1 -2190.994,E2 -2190.994} C_VEL
LIN {X 0,Y 573.245,Z 343.7,A -85,B 0,C 180,E1 -2193.52,E2 -2193.52} C_VEL
LIN {X 0,Y 573.181,Z 343.716,A -85,B 0,C 180,E1 -2196.054,E2 -2196.054} C_VEL
LIN {X 0,Y 573.229,Z 343.702,A -85,B 0,C 180,E1 -2198.703,E2 -2198.703} C_VEL
LIN {X 0,Y 573.186,Z 343.709,A -85,B 0,C 180,E1 -2201.587,E2 -2201.587} C_VEL
LIN {X 0,Y 573.203,Z 343.709,A -85,B 0,C 180,E1 -2204.336,E2 -2204.336} C_VEL
LIN {X 0,Y 573.207,Z 343.705,A -85,B 0,C 180,E1 -2207.362,E2 -2207.362} C_VEL
LIN {X 0,Y 573.222,Z 343.704,A -85,B 0,C 180,E1 -2210.571,E2 -2210.571} C_VEL
LIN {X 0,Y 573.201,Z 343.705,A -85,B 0,C 180,E1 -2213.073,E2 -2213.073} C_VEL
LIN {X 0,Y 573.241,Z 343.707,A -85,B 0,C 180,E1 -2215.669,E2 -2215.669} C_VEL
LIN {X 0,Y 573.216,Z 343.709,A -85,B 0,C 180,E1 -2218.182,E2 -2218.182} C_VEL
LIN {X 0,Y 573.221,Z 343.704,A -85,B 0,C 180,E1 -2220.631,E2 -2220.631} C_VEL
LIN {X 0,Y 573.243,Z 343.846,A -85,B 0,C 180,E1 -2223.644,E2 -2223.644} C_VEL
LIN {X 0,Y 574.607,Z 349.975,A -85,B 0,C 180,E1 -2224.459,E2 -2224.459} C_VEL
LIN {X 0,Y 574.401,Z 370.263,A -85,B 0,C 180,E1 -2226.949,E2 -2226.949} C_VEL
LIN {X 0,Y 574.05,Z 395.233,A -85,B 0,C 180,E1 -2229.952,E2 -2229.952} C_VEL
LIN {X 0,Y 574.016,Z 398.864,A -85,B 0,C 180,E1 -2230.384,E2 -2230.384} C_VEL
LIN {X 0,Y 575.18,Z 405.388,A -85,B 0,C 180,E1 -2230.516,E2 -2230.516} C_VEL
LIN {X 0,Y 574.765,Z 564.975,A -85,B 0,C 180,E1 -2232.579,E2 -2232.579} C_VEL
LIN {X 0,Y 574.628,Z 580.674,A -85,B 0,C 180,E1 -2232.93,E2 -2232.93} C_VEL
LIN {X 0,Y 574.429,Z 596.018,A -85,B 0,C 180,E1 -2233.427,E2 -2233.427} C_VEL
LIN {X 0,Y 574.293,Z 609.751,A -85,B 0,C 180,E1 -2234.016,E2 -2234.016} C_VEL
LIN {X 0,Y 574.05,Z 623.228,A -85,B 0,C 180,E1 -2234.738,E2 -2234.738} C_VEL
LIN {X 0,Y 573.863,Z 636.804,A -85,B 0,C 180,E1 -2235.631,E2 -2235.631} C_VEL
LIN {X 0,Y 573.636,Z 649.338,A -85,B 0,C 180,E1 -2236.628,E2 -2236.628} C_VEL
LIN {X 0,Y 573.478,Z 659.74,A -85,B 0,C 180,E1 -2237.615,E2 -2237.615} C_VEL
LIN {X 0,Y 573.287,Z 669.763,A -85,B 0,C 180,E1 -2238.733,E2 -2238.733} C_VEL
LIN {X 0,Y 573.244,Z 678.851,A -85,B 0,C 180,E1 -2239.938,E2 -2239.938} C_VEL
LIN {X 0,Y 573.133,Z 686.728,A -85,B 0,C 180,E1 -2241.182,E2 -2241.182} C_VEL
LIN {X 0,Y 573.075,Z 694.085,A -85,B 0,C 180,E1 -2242.601,E2 -2242.601} C_VEL
LIN {X 0,Y 573.042,Z 699.92,A -85,B 0,C 180,E1 -2244.015,E2 -2244.015} C_VEL
LIN {X 0,Y 572.951,Z 703.382,A -85,B 0,C 180,E1 -2245.073,E2 -2245.073} C_VEL
LIN {X 0,Y 573.005,Z 706.887,A -85,B 0,C 180,E1 -2246.483,E2 -2246.483} C_VEL
LIN {X 0,Y 572.938,Z 709.191,A -85,B 0,C 180,E1 -2247.89,E2 -2247.89} C_VEL
LIN {X 0,Y 572.936,Z 710.349,A -85,B 0,C 180,E1 -2249.296,E2 -2249.296} C_VEL
LIN {X 0,Y 572.936,Z 710.349,A -85,B 0,C 180,E1 -2250.702,E2 -2250.702} C_VEL
LIN {X 0,Y 572.938,Z 709.192,A -85,B 0,C 180,E1 -2252.108,E2 -2252.108} C_VEL
LIN {X 0,Y 573.005,Z 706.889,A -85,B 0,C 180,E1 -2253.515,E2 -2253.515} C_VEL
LIN {X 0,Y 572.951,Z 703.388,A -85,B 0,C 180,E1 -2254.925,E2 -2254.925} C_VEL
LIN {X 0,Y 573.013,Z 698.613,A -85,B 0,C 180,E1 -2256.336,E2 -2256.336} C_VEL
